	IF IP_C.ERROR > DWORD#0 AND IP_C.C_ENABLE AND NOT IP_C.TIME_RESET THEN  (* IP Control 1 *)
		IF ip_c_red_disable = FALSE OR IP_C.ERROR <> DWORD#16#FD000000 THEN
			ERROR_C := IP_C.ERROR;
			ERROR_T := BYTE#2;
			step := 980;
		END_IF;
	END_IF;

	IF FSD.MODE = BYTE#0 THEN
		IF FSD.ERROR > BYTE#0 THEN
			ERROR_C := BYTE_TO_DWORD(FSD.ERROR);
			ERROR_T := BYTE#4; (* Dateizugriff *)
			step := 980;
		END_IF;
	END_IF;
END_IF;

IF TON_WAIT.Q THEN (* Ablaufstörung - Schrittkette *)
	ERROR_C := SHL(INT_TO_DWORD(step),16) OR INT_TO_DWORD(rcv_state); (* aktuellen Schritt und letzten SMTP Status eintragen *)
	ERROR_T := BYTE#5;
	step := 980;
END_IF;

(* ######################################################## *)

DNS_CLIENT(IP_C:=IP_C, S_BUF:=S_BUF, R_BUF:=R_BUF, DOMAIN:=URL_DATA.DOMAIN, IP4_DNS:= DNS_IP4, ACTIVATE:=step=10); (* DNS-Client *)
IPC(IP:= DWORD#0, PORT:= WORD#0 , TIME_OUT:= TIMEOUT, IP_C:= IP_C, S_BUF:= S_BUF, R_BUF:= R_BUF); (* SMTP Steuerkanal *)
FS(FSD:=FSD,PT:=F_BUF); (* FILE_SERVER *)
BASE64_ENCODE_STR(RUN:= b64_start, STR1:= b64_str1, STR2:= b64_str2, DONE=> b64_done); (* BASE64 kodierung *)

TON_WAIT(IN:=step = last_step AND step > 0,PT:=timeout2);
last_step := step;
activate_last := ACTIVATE;
BUSY := step <> 0;

(* revision history
ks	01. jan. 2011	rev 1.0
	original version
ks	06. apr. 2011	rev 1.1
	list_len und list_get durch element_count und element_get ersetzt
ks	11. may 2011	rev 1.2
	ip_control - remote disconnect error ausblenden, und sonderbehandlung für pcworx
ks	30. may 2011	rev 1.3
	fehler bei receive-timeout
ks	05. may. 2012	rev 1.4
	FileServer AutoClose entfernt und Fehler im Alias Name korrigiert
ks	06. apr. 2013	rev 1.5
	Fehler bei Authorisierungsabfrage bei 1&1 Provider behoben
ks	22. feb. 2016	rev 1.6
	integration SSL/TLS
ks	11. aug. 2016	rev 1.7
	bugfix: Find SSL/TLS String in URL_DATA.PROTOCOL
*)

END_FUNCTION_BLOCK

// POUs/CONVERT/MD5_CRAM_AUTH
FUNCTION_BLOCK MD5_CRAM_AUTH
VAR_IN_OUT
	RUN : BOOL;
	USERNAME : STRING(64);
	PASSWORD : STRING(64);
	B64_TS : STRING(64);  (* Base64 coded ServerTimeStamp *)
	AUTH_KEY : STRING(192);
END_VAR
VAR
	BASE64_DECODE_STR : BASE64_DECODE_STR;
	BASE64_ENCODE_STR : BASE64_ENCODE_STR;
	MD5_STREAM : MD5_STREAM;
	step : INT;
	md5_mode : INT;
	buf : ARRAY [0..63] OF BYTE;
	md5 : ARRAY [0..15] OF BYTE;
	md5_first : ARRAY [0..15] OF BYTE;
	md5_str1 : STRING(64);
	md5_str2 : STRING(64);
	size : UDINT;
	n1 : INT;
	n2 : INT;
	pos : UDINT;
	b64d_run : BOOL;
	b64d_done : BOOL;
	b64e_run : BOOL;
	b64e_done : BOOL;
	str_192 : STRING(192);
	str_144 : STRING(144);
	xpad : BYTE;
	pt : POINTER TO BYTE;
END_VAR

(*
version 1.0		10. may 2010
programmer 	ks
tested by		ks

Der Baustein MD5_CRAM_AUTH (Challenge-Response Authentication Mechanism, Message Digest 5) benutzt
das Authentifizierungsverfahren nach dem Challenge-Response-Prinzip auf der Basis des MD5-HMAC-Algorithmus.
Es wird beispielsweise zur Authentifizierung gegenüber SMTP- oder IMAP-Servern eingesetzt, da es die Übertragung des Passworts im Klartext vermeidet.
Durch dieses Verfahren kann auch über unverschlüsselte Kanäle eine sichere Authentifizierung gegenüber einem Server erfolgen


*)

CASE step OF

0:	IF RUN THEN
		step := 5;
		str_192 := B64_TS;
		b64d_run := TRUE;
	END_IF;

5: IF B64D_DONE THEN (* IPAD Zyklus *)
		b64d_run := FALSE;
		xpad := 16#36;
		md5_str1 := PASSWORD;
		md5_str2 := str_144;
		size := 64 + LEN(md5_str2);
		md5_mode := 1;
		step := 10;
	END_IF;

10: IF md5_mode = 3 THEN (* OPAD Zyklus *)
		md5_first := md5; (* md5 array vom IPAD sichern *)
		xpad := 16#5C;
		size := 64 + 16;
		md5_mode := 1;
		step := 20;
	END_IF;

20: IF md5_mode = 3 THEN
		md5_mode := 0;
		str_144 := CONCAT(USERNAME , ' ');
		str_144 := CONCAT(str_144 , MD5_TO_STRH(md5));
		b64e_run := TRUE;
		step := 30;
	END_IF;

30: IF B64E_DONE THEN
		AUTH_KEY := str_192;
		b64e_run := FALSE;
		RUN := FALSE;
		step := 0; (* alles beendet !! *)
	END_IF;

END_CASE;

(* ----------- md5 -------------- *)
CASE md5_mode OF

1:	n2 := LEN(md5_str1) - 1;
	pt := ADR(md5_str1);
	FOR n1 := 0 TO n2 DO (* string in buf kopieren *)
		buf[n1] := pt^ XOR xpad;
		pt := pt + 1;
	END_FOR;
	FOR n1 := n2 + 1 TO 63 DO (* mit ipad füllen *)
		buf[n1] := xpad;
	END_FOR;

2:	(* Data copy and Calc *)
	IF size > 0 AND pos >= 64 THEN
		IF step = 20 THEN
			FOR n1 := 0 TO 15 DO
				buf[n1] := md5_first[n1];
			END_FOR;
		ELSE
			n2 := LEN(md5_str2) - 1;
			pt := ADR(md5_str2);
			FOR n1 := 0 TO n2 DO (* string in buf kopieren *)
				buf[n1] := pt^;
				pt := pt + 1;
			END_FOR;
		END_IF;
	END_IF;

END_CASE;

IF md5_mode > 0 THEN
	MD5_STREAM(SIZE:=size, MODE:=md5_mode, BUF:=buf, MD5:=md5, POS=>pos);
END_IF;

BASE64_DECODE_STR(RUN:=b64d_run, STR1:=str_192, STR2:=str_144, DONE=>b64d_done);
BASE64_ENCODE_STR(RUN:=b64e_run, STR1:=str_144, STR2:=str_192, DONE=>b64e_done);

(* revision history

hm		10. mai. 2010	rev 1.0
	original version
*)

END_FUNCTION_BLOCK

// POUs/CONVERT/MD5_TO_STRH
FUNCTION MD5_TO_STRH : STRING(32)
VAR_INPUT
	MD5 : ARRAY [0..15] OF BYTE;
END_VAR
VAR
	i : INT;
	tmp : BYTE;
	pt : POINTER TO BYTE;
END_VAR
(*
version 1.0	06. dec. 2009
programmer 	ks
tested BY	ks

MD5_TO_STRH konvertiert das MD5 Hash Array in einen HEX-String
*)

pt := ADR(MD5_TO_STRH); (* read output adress to pointer *)

FOR i := 0 TO 15 DO; (* write the 8 hex characters backwards *)
	tmp := SHR(MD5[i],4);
	PT^ := tmp + SEL(tmp <= 9,87,48);
	pt := pt + 1; (* decrement the pointer *)
	tmp := MD5[i] AND 2#1111;
	PT^ := tmp + SEL(tmp <= 9,87,48);
	pt := pt + 1; (* decrement the pointer *)
END_FOR;
pt^:= 0; (* write the closing byte for the string *)

(* revision history

ks	6. dec. 2009 rev 1.0
	original version

*)

END_FUNCTION

// POUs/CONVERT/MD5_STREAM
FUNCTION_BLOCK MD5_STREAM
VAR_IN_OUT
	MODE : INT;
	BUF : ARRAY [0..63] OF BYTE;
	MD5 : ARRAY [0..15] OF BYTE;
	SIZE : UDINT;
END_VAR

VAR_OUTPUT
	POS : UDINT;
END_VAR

VAR
	hash : ARRAY [0..3] OF DWORD;
	a : DWORD;
	b : DWORD;
	c : DWORD;
	d : DWORD;
	end : UDINT;
	block : UDINT;
	x : ARRAY [0..15] OF DWORD;
	n : INT;
	n1 : INT;
	z : INT;
	pad_1 : BOOL;
END_VAR

(*
version 1.0	06. dec. 2009
programmer 	ks
tested BY	ks

MD5_STREAM berechnet den MD5 Hash eines Datenstromes
*)

CASE MODE OF

1:	(* Initialisierung der Hash-Werte *)
	hash[0] := DWORD#16#67452301;
	hash[1] := DWORD#16#EFCDAB89;
	hash[2] := DWORD#16#98BADCFE;
	hash[3] := DWORD#16#10325476;

	block := SHR(SIZE,6) + BOOL_TO_UDINT((UDINT_TO_BYTE(SIZE) AND 16#3F) > 55);
	pad_1 := FALSE;
	POS := 0;
	End := SIZE;
	SIZE := MIN(64,End);
	MODE := 2;

2:	(* Fuell-Bytes anhängen *)
	FOR n := UDINT_TO_INT(SIZE) TO 63 DO
		BUF[n] := 0;
	END_FOR;

	IF SIZE < 64 AND NOT pad_1 THEN
		BUF[SIZE] := 2#1000_0000;
		pad_1 := TRUE;
	END_IF;

	POS := POS + SIZE;
	SIZE := MIN(64,End - POS);

	n := 0;	(* Byte-Array in DWORD-Array umkopieren *)
	FOR n1 := 0 TO 15 DO
		x[n1] := OSCAT_BASIC.DWORD_OF_BYTE(BUF[n+3],BUF[n+2],BUF[n+1],BUF[n]); (* Little Endian Format *)
		n := n + 4;
	END_FOR;

	IF block = 0 THEN (* am Ende des letzten Blocks die Datenlänge eintragen *)
		x[14] := SHL(UDINT_TO_DWORD(End),3); (* Anzahl Datenbits im Little-Endian Format eintragen *)
		MODE := 3;
	ELSE
		block := block - 1;
	END_IF;

	a := hash[0];
	b := hash[1];
	c := hash[2];
	d := hash[3];

	a := MD5_AUX(1, a, b, c, d, X[00], 07, 16#D76AA478); (* 01 *)
	d := MD5_AUX(1, d, a, b, c, X[01], 12, 16#E8C7B756); (* 02 *)
	c := MD5_AUX(1, c, d, a, b, X[02], 17, 16#242070DB); (* 03 *)
	b := MD5_AUX(1, b, c, d, a, X[03], 22, 16#C1BDCEEE); (* 04 *)
	a := MD5_AUX(1, a, b, c, d, X[04], 07, 16#F57C0FAF); (* 05 *)
	d := MD5_AUX(1, d, a, b, c, X[05], 12, 16#4787C62A); (* 06 *)
	c := MD5_AUX(1, c, d, a, b, X[06], 17, 16#A8304613); (* 07 *)
	b := MD5_AUX(1, b, c, d, a, X[07], 22, 16#FD469501); (* 08 *)
	a := MD5_AUX(1, a, b, c, d, X[08], 07, 16#698098D8); (* 09 *)
	d := MD5_AUX(1, d, a, b, c, X[09], 12, 16#8B44F7AF); (* 10 *)
	c := MD5_AUX(1, c, d, a, b, X[10], 17, 16#FFFF5BB1); (* 11 *)
	b := MD5_AUX(1, b, c, d, a, X[11], 22, 16#895CD7BE); (* 12 *)
	a := MD5_AUX(1, a, b, c, d, X[12], 07, 16#6B901122); (* 13 *)
	d := MD5_AUX(1, d, a, b, c, X[13], 12, 16#FD987193); (* 14 *)
	c := MD5_AUX(1, c, d, a, b, X[14], 17, 16#A679438E); (* 15 *)
	b := MD5_AUX(1, b, c, d, a, X[15], 22, 16#49B40821); (* 16 *)

	a := MD5_AUX(2, a, b, c, d, X[01], 05, 16#F61E2562); (* 17 *)
	d := MD5_AUX(2, d, a, b, c, X[06], 09, 16#C040B340); (* 18 *)
	c := MD5_AUX(2, c, d, a, b, X[11], 14, 16#265E5A51); (* 19 *)
	b := MD5_AUX(2, b, c, d, a, X[00], 20, 16#E9B6C7AA); (* 20 *)
	a := MD5_AUX(2, a, b, c, d, X[05], 05, 16#D62F105D); (* 21 *)
	d := MD5_AUX(2, d, a, b, c, X[10], 09, 16#02441453); (* 22 *)
	c := MD5_AUX(2, c, d, a, b, X[15], 14, 16#D8A1E681); (* 23 *)
	b := MD5_AUX(2, b, c, d, a, X[04], 20, 16#E7D3FBC8); (* 24 *)
	a := MD5_AUX(2, a, b, c, d, X[09], 05, 16#21E1CDE6); (* 25 *)
	d := MD5_AUX(2, d, a, b, c, X[14], 09, 16#C33707D6); (* 26 *)
	c := MD5_AUX(2, c, d, a, b, X[03], 14, 16#F4D50D87); (* 27 *)
	b := MD5_AUX(2, b, c, d, a, X[08], 20, 16#455A14ED); (* 28 *)
	a := MD5_AUX(2, a, b, c, d, X[13], 05, 16#A9E3E905); (* 29 *)
	d := MD5_AUX(2, d, a, b, c, X[02], 09, 16#FCEFA3F8); (* 30 *)
	c := MD5_AUX(2, c, d, a, b, X[07], 14, 16#676F02D9); (* 31 *)
	b := MD5_AUX(2, b, c, d, a, X[12], 20, 16#8D2A4C8A); (* 32 *)

	a := MD5_AUX(3, a, b, c, d, X[05], 04, 16#FFFA3942); (* 33 *)
	d := MD5_AUX(3, d, a, b, c, X[08], 11, 16#8771F681); (* 34 *)
	c := MD5_AUX(3, c, d, a, b, X[11], 16, 16#6D9D6122); (* 35 *)
	b := MD5_AUX(3, b, c, d, a, X[14], 23, 16#FDE5380C); (* 36 *)
	a := MD5_AUX(3, a, b, c, d, X[01], 04, 16#A4BEEA44); (* 37 *)
	d := MD5_AUX(3, d, a, b, c, X[04], 11, 16#4BDECFA9); (* 38 *)
	c := MD5_AUX(3, c, d, a, b, X[07], 16, 16#F6BB4B60); (* 39 *)
	b := MD5_AUX(3, b, c, d, a, X[10], 23, 16#BEBFBC70); (* 40 *)
	a := MD5_AUX(3, a, b, c, d, X[13], 04, 16#289B7EC6); (* 41 *)
	d := MD5_AUX(3, d, a, b, c, X[00], 11, 16#EAA127FA); (* 42 *)
	c := MD5_AUX(3, c, d, a, b, X[03], 16, 16#D4EF3085); (* 43 *)
	b := MD5_AUX(3, b, c, d, a, X[06], 23, 16#04881D05); (* 44 *)
	a := MD5_AUX(3, a, b, c, d, X[09], 04, 16#D9D4D039); (* 45 *)
	d := MD5_AUX(3, d, a, b, c, X[12], 11, 16#E6DB99E5); (* 46 *)
	c := MD5_AUX(3, c, d, a, b, X[15], 16, 16#1FA27CF8); (* 47 *)
	b := MD5_AUX(3, b, c, d, a, X[02], 23, 16#C4AC5665); (* 48 *)

	a := MD5_AUX(4, a, b, c, d, X[00], 06, 16#F4292244); (* 49 *)
	d := MD5_AUX(4, d, a, b, c, X[07], 10, 16#432AFF97); (* 50 *)
	c := MD5_AUX(4, c, d, a, b, X[14], 15, 16#AB9423A7); (* 51 *)
	b := MD5_AUX(4, b, c, d, a, X[05], 21, 16#FC93A039); (* 52 *)
	a := MD5_AUX(4, a, b, c, d, X[12], 06, 16#655B59C3); (* 53 *)
	d := MD5_AUX(4, d, a, b, c, X[03], 10, 16#8F0CCC92); (* 54 *)
	c := MD5_AUX(4, c, d, a, b, X[10], 15, 16#FFEFF47D); (* 55 *)
	b := MD5_AUX(4, b, c, d, a, X[01], 21, 16#85845DD1); (* 56 *)
	a := MD5_AUX(4, a, b, c, d, X[08], 06, 16#6FA87E4F); (* 57 *)
	d := MD5_AUX(4, d, a, b, c, X[15], 10, 16#FE2CE6E0); (* 58 *)
	c := MD5_AUX(4, c, d, a, b, X[06], 15, 16#A3014314); (* 59 *)
	b := MD5_AUX(4, b, c, d, a, X[13], 21, 16#4E0811A1); (* 60 *)
	a := MD5_AUX(4, a, b, c, d, X[04], 06, 16#F7537E82); (* 61 *)
	d := MD5_AUX(4, d, a, b, c, X[11], 10, 16#BD3AF235); (* 62 *)
	c := MD5_AUX(4, c, d, a, b, X[02], 15, 16#2AD7D2BB); (* 63 *)
	b := MD5_AUX(4, b, c, d, a, X[09], 21, 16#EB86D391); (* 64 *)

	hash[0] := hash[0] + a;
	hash[1] := hash[1] + b;
	hash[2] := hash[2] + c;
	hash[3] := hash[3] + d;

END_CASE;

IF MODE = 3 THEN
	z := 0;
	FOR n := 0 TO 3 DO (* von Little-Endian auf Big-Endian format konvertieren und DWORD auf BYTE-Array *)
		FOR n1 := 0 TO 3 DO
			MD5[z] := DWORD_TO_BYTE(hash[n]);
			hash[n] := ROR(hash[n],8);
			z := z + 1;
		END_FOR;
	END_FOR;
END_IF;

(* revision history

ks	6. dec. 2009 rev 1.0
	original version

*)

END_FUNCTION_BLOCK

// POUs/CONVERT/MD5_AUX
FUNCTION MD5_AUX : DWORD
VAR_INPUT
	N : INT;
	A : DWORD;
	B : DWORD;
	C : DWORD;
	D : DWORD;
	X : DWORD;
	U : INT;
	T : DWORD;
END_VAR
VAR
	w : DWORD;
END_VAR

(*
version 1.0	06. dec. 2009
programmer 	ks
tested by	ks

MD5_AUX ist ein Zusatzbaustein füR MD5_STREAM und enthäLT wiederkehrende Berechnungen
*)

CASE N OF
	1: w := (B AND C) OR (NOT(B) AND D);
	2: w := (B AND D) OR (C AND NOT D);
	3: w := (B XOR C XOR D);
	4: w := (C XOR (B OR  NOT(D)));
END_CASE

MD5_AUX := B + ROL(A + w + X + T,U);

(* revision history

ks	6. dec. 2009 rev 1.0
	original version

*)

END_FUNCTION

// POUs/DEMO/DLOG_FILE_HTML_DEMO
PROGRAM DLOG_FILE_HTML_DEMO
VAR
	cur_dt: DT;
	enable: BOOL := TRUE;
	trig_t : TIME := T#5s;
	trig_m : BOOL;
	error_c: DWORD;
	error_t: BYTE;
	auto_close: TIME := T#10s;

	x1: DLOG_DT;
	x2 : DLOG_REAL;
	x3 : DLOG_DINT;
	x4 : DLOG_BOOL;
	x5: DLOG_STRING;
	x : DLOG_DATA;
	RTC_2: oscat_basic.RTC_2;
	DLOG_STORE_FILE_HTML: DLOG_STORE_FILE_HTML;
	GEN_SIN_1: oscat_basic.GEN_SIN;
	COUNT_DR: oscat_basic.COUNT_DR;

	html_caption: STRING := 'Das ist der Titel';
	html_tr_even: STRING := 'BGCOLOR=#B3B7FF';
	html_tr_odd: STRING := 'BGCOLOR=#E0E0E0';
	html_tr_head: STRING := 'BGCOLOR=#FFFF40';
	html_table : STRING := 'BORDER="1"';
END_VAR

VAR RETAIN
	save_data : DLOG_SAVE;
END_VAR
VAR // added by the converter: edge detectors and wires of the graphical bodies
    _w1 : ANY;
END_VAR

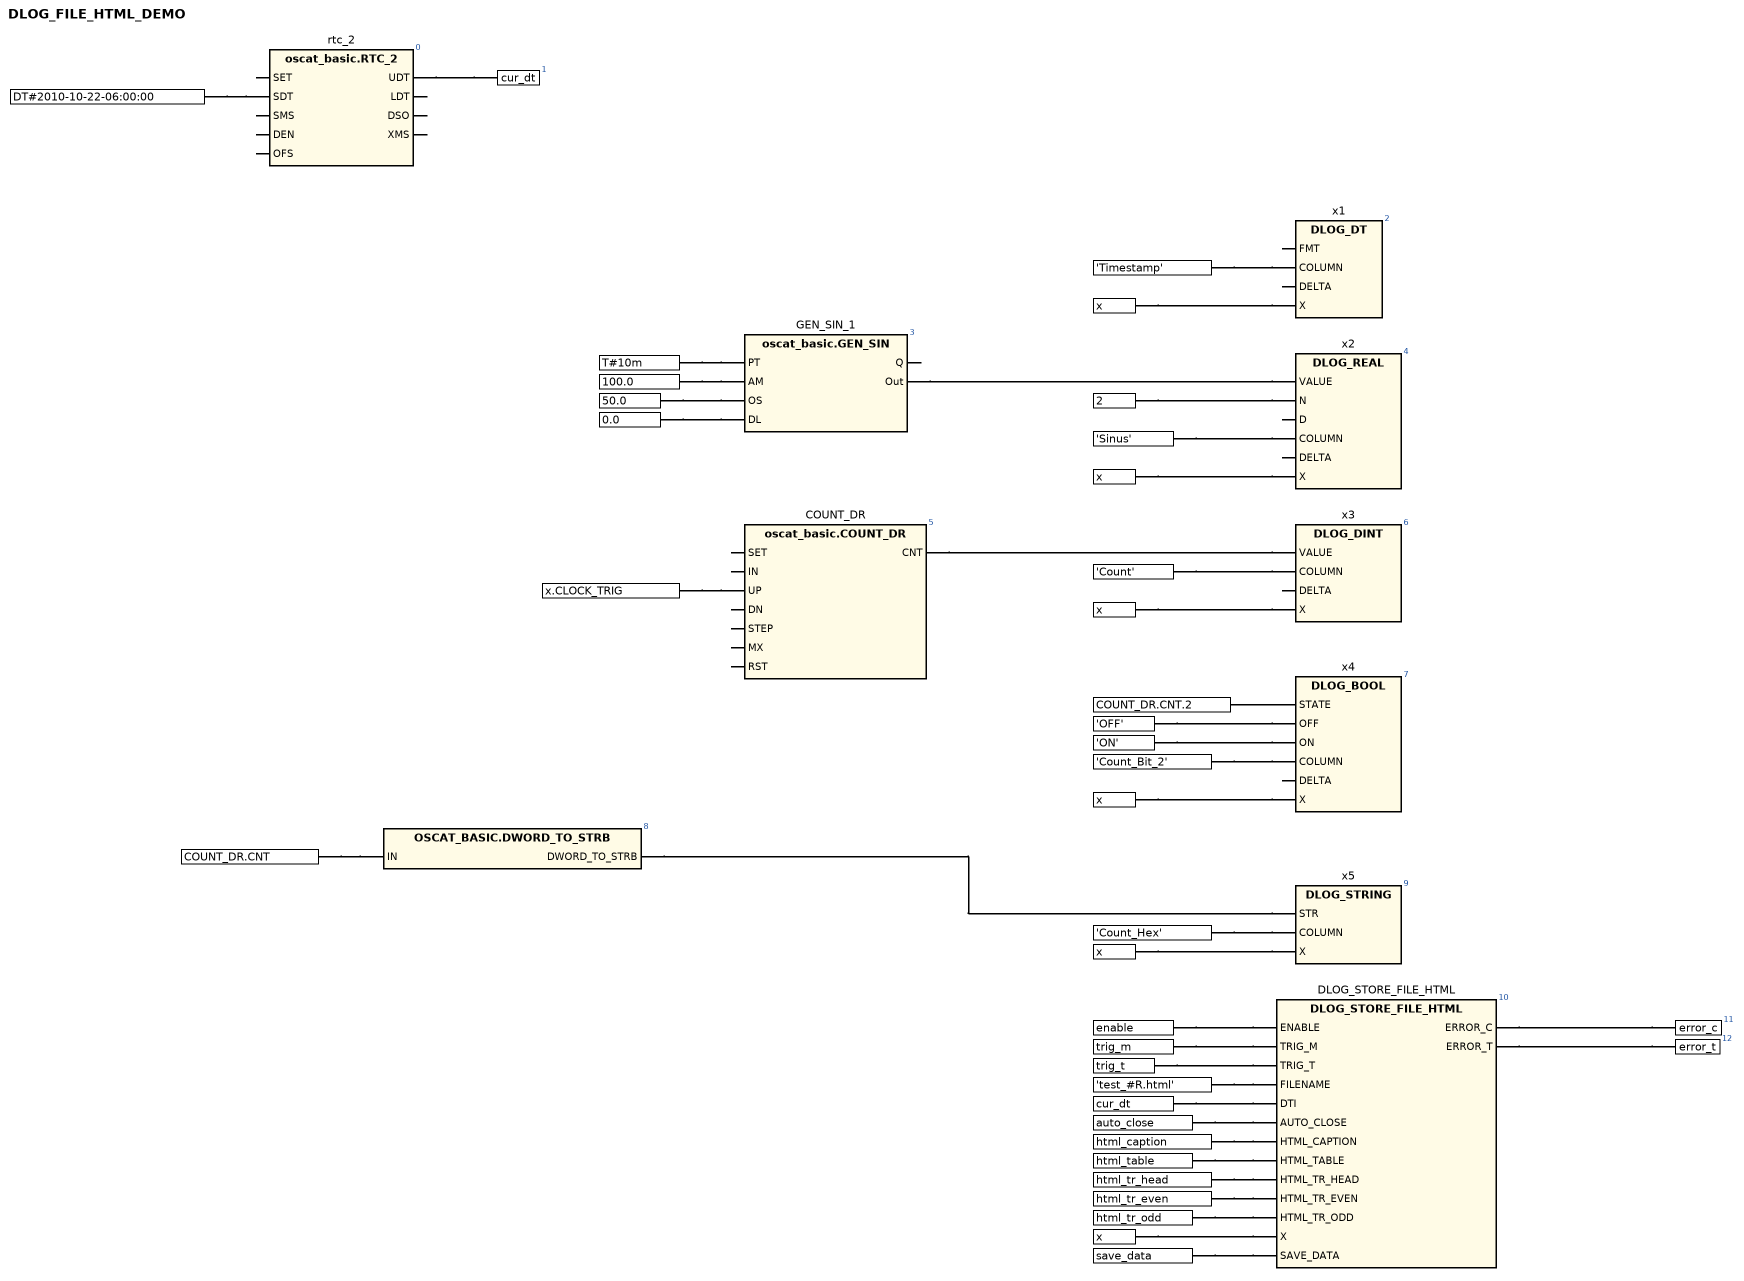
rtc_2(SDT := DT#2010-10-22-06:00:00); // oscat_basic.RTC_2
cur_dt := rtc_2.UDT;
x1(COLUMN := 'Timestamp', X := x); // DLOG_DT
GEN_SIN_1(PT := T#10m, AM := 100.0, OS := 50.0, DL := 0.0); // oscat_basic.GEN_SIN
x2(VALUE := GEN_SIN_1.Out, N := 2, COLUMN := 'Sinus', X := x); // DLOG_REAL
COUNT_DR(UP := x.CLOCK_TRIG); // oscat_basic.COUNT_DR
x3(VALUE := COUNT_DR.CNT, COLUMN := 'Count', X := x); // DLOG_DINT
x4(STATE := COUNT_DR.CNT.2, OFF := 'OFF', ON := 'ON', COLUMN := 'Count_Bit_2', X := x); // DLOG_BOOL
_w1 := OSCAT_BASIC.DWORD_TO_STRB(IN := COUNT_DR.CNT);
x5(STR := _w1, COLUMN := 'Count_Hex', X := x); // DLOG_STRING
DLOG_STORE_FILE_HTML(
    ENABLE := enable,
    TRIG_M := trig_m,
    TRIG_T := trig_t,
    FILENAME := 'test_#R.html',
    DTI := cur_dt,
    AUTO_CLOSE := auto_close,
    HTML_CAPTION := html_caption,
    HTML_TABLE := html_table,
    HTML_TR_HEAD := html_tr_head,
    HTML_TR_EVEN := html_tr_even,
    HTML_TR_ODD := html_tr_odd,
    X := x,
    SAVE_DATA := save_data);
error_c := DLOG_STORE_FILE_HTML.ERROR_C;
error_t := DLOG_STORE_FILE_HTML.ERROR_T;

END_PROGRAM

// POUs/DATA_LOG/DLOG_STORE_FILE_HTML
FUNCTION_BLOCK DLOG_STORE_FILE_HTML
VAR_IN_OUT
	X : DLOG_DATA;
	SAVE_DATA : DLOG_SAVE;
END_VAR
VAR_INPUT
	ENABLE : BOOL;
	TRIG_M : BOOL;
	TRIG_T : TIME;
	FILENAME : STRING;
	DTI : DT;
	AUTO_CLOSE : TIME := T#15s;
	HTML_CAPTION : STRING;
	HTML_TABLE : STRING;
	HTML_TR_HEAD : STRING;
	HTML_TR_EVEN : STRING;
	HTML_TR_ODD : STRING;
END_VAR
VAR_OUTPUT
	ERROR_C : DWORD;
	ERROR_T : BYTE;
END_VAR
VAR
	FS : FILE_SERVER;
	FSD : FILE_SERVER_DATA;
	PT : NETWORK_BUFFER;
	UCB : UNI_CIRCULAR_BUFFER;
	trig_auto : BOOL;
	trig_stored : BOOL;
	trig_tmp : BOOL;
	trig_m_last : BOOL;
	dti_last : DT := DT#2070-02-06-06:28:15;
	fn_last : STRING;
	str : STRING(OSCAT_BASIC.STRING_LENGTH);
	fn : STRING;
	step_1 : INT;
	step_2 : INT;
	idx : INT;
	log_state : USINT;
	log_stop : BOOL;
	n : INT;
	wd_ton : TON;
	wd_time : TIME;
	aw_ton : TON;
	aw_enable : BOOL;
	aw_aktiv : BOOL;
	total_bytes : UDINT;
	cur_ode : BYTE;

	(*
	LOG_MSG : LOG_MSG;
	_debug_enable : BOOL := TRUE;
	*)

END_VAR

(*
version 1.3		21. mar. 2016
programmer		ks
tested by			ks

DLOG_STORE_FILE_HTML schreibt die DLOG Parameter in einen lokale Datei im HMTL-Format 

*)

X.DTI := DTI; (* Datum / Zeit eintragen *)
X.CLOCK_TRIG := DTI <> dti_last;
dti_last := DTI;
trig_auto := FALSE;
IF X.CLOCK_TRIG THEN (* Impuls in jeder Sekunde *)
	fn := OSCAT_BASIC.DT_TO_STRF(DTI, 0, FILENAME, 0); (* automatische Dateinamen generierung *)
	IF TRIG_T >= T#1000ms THEN (* automatischer Trigger *)
		trig_auto := DT_TO_UDINT(DTI) MOD (TIME_TO_UDINT(TRIG_T) / UDINT#1000) = UDINT#0;
	END_IF;
END_IF;

CASE step_1 OF

00:	IF ENABLE THEN
		aw_enable := AUTO_CLOSE >= T#5s;
		wd_time := SEL(X.LOAD_TIME_MAX > T#0s, T#5ms,X.LOAD_TIME_MAX);
		fn_last := fn; (* aktuellen Dateinnamen speichern *)
		IF X.ID_MAX = USINT#0 THEN (* nur einmal nach Satellitenbausteinen scannen *)
			X.ADD_COM := 01; (* ADD INFO *)
			X.STORE_TYPE := BYTE#4; (* HTML-Modus *)
		END_IF;
		step_1 := 10;

		(* ---------------- Debug-Message -----------------------*)
		(*IF _debug_enable THEN
			LOG_CL.NEW_MSG := 'FILE_HTML1 - Start: File [~1], [~2]';
			LOG_CL.PRINTF[1] := fn_last;
			LOG_CL.PRINTF[2] := DT_TO_STRING(DTI);
			LOG_MSG();
		END_IF;*)
		(* -----------------------------------------------------------------*)

	END_IF;

10:	X.UCB.D_STRING := fn_last;
	IF fn_last = SAVE_DATA.FN_REM THEN
		X.UCB.D_HEAD := WORD#16#F201; (* Filemode open + write *)
		X.ADD_COM := 00;
	ELSE
		X.UCB.D_HEAD := WORD#16#F301; (* Filemode create + write *)
		X.ADD_COM := 02; (* ADD HEADER *)
	END_IF;

	X.UCB.D_MODE := 1; (* Dateinamen als String ablegen *)
	UCB(DATA:=X.UCB); (* Daten eintragen *)
	step_1 := 30;

30:	(* LOG-Trigger verarbeiten *)
	trig_tmp := (TRIG_M AND NOT trig_m_last) OR trig_auto OR X.ADD_DATA_REQ;

	IF ENABLE = FALSE OR fn <> fn_last THEN (* ENABLE = 0 oder neuen Dateinamen -> Log Stop *)
		trig_stored := trig_tmp; (* aktuellen Triggerpuls speichern *)
		X.UCB.D_HEAD := WORD#16#EE00;
		X.UCB.D_MODE := 1;
		UCB(DATA:=X.UCB); (* Element schreiben *)
		X.ADD_COM := 00;
		step_1 := 00;

		(* ---------------- Debug-Message -----------------------*)
		(*IF _debug_enable THEN
			LOG_CL.NEW_MSG := 'FILE_HTML1 - Stop: [~2]';
			LOG_CL.PRINTF[2] := DT_TO_STRING(DTI);
			LOG_MSG();
		END_IF;*)
		(* -----------------------------------------------------------------*)

	ELSIF ENABLE THEN
		IF trig_tmp OR trig_stored THEN (* manueller, automatischer oder externer Trigger *)
			trig_stored := FALSE;
			X.ADD_COM := 03; (* ADD DATA *)
			SAVE_DATA.TRIG_CNT := SAVE_DATA.TRIG_CNT + UDINT#1;
			SAVE_DATA.TRIG_CNT_TOTAL  := SAVE_DATA.TRIG_CNT_TOTAL + UDINT#1;
			(* ---------------- Debug-Message -----------------------*)
			(*IF _debug_enable THEN
				LOG_CL.NEW_MSG := 'FILE_HTML1 - Trig: [~2]';
				LOG_CL.PRINTF[2] := DT_TO_STRING(DTI);
				LOG_MSG();
			END_IF;*)
			(* -----------------------------------------------------------------*)
		ELSE
			X.ADD_COM := 04;	(* ADD DATA REQ *)
		END_IF;
	END_IF;

END_CASE;
X.ADD_DATA_REQ := FALSE; (* externe Anforderung rücksetzen *)

(* ##################################### *)

CASE step_2 OF

00:	aw_ton(IN:= idx > 0 AND aw_enable , PT:= AUTO_CLOSE); (* AutoWrite Timer *)
	IF aw_ton.Q THEN (* Zeitgesteuertes Datenschreiben *)
		aw_aktiv := TRUE;
		step_2 := 10; (* Daten schreiben *)
		(* ---------------- Debug-Message -----------------------*)
		(*IF _debug_enable THEN
			LOG_CL.NEW_MSG := 'FILE_HTML2 - AutoWrite: [~2]';
			LOG_CL.PRINTF[2] := DT_TO_STRING(DTI);
			LOG_MSG();
		END_IF;*)
		(* -----------------------------------------------------------------*)

	ELSE
		wd_ton(IN:= FALSE, PT:= wd_time);
		wd_ton(IN:= TRUE);
		WHILE X.UCB.BUF_COUNT > 0 AND step_2 = 0 AND wd_ton.Q = FALSE DO

			X.UCB.D_MODE := 10;
			UCB(DATA:=X.UCB); (* Element lesen , aber noch nicht entfernen *)

			IF X.UCB.D_HEAD > WORD#16#F000 THEN (* F301 oder F201 *)

				str := CONCAT('<html><body><table ',HTML_TABLE);
		        		str := CONCAT(str,'><caption>');
		        		str := CONCAT(str,HTML_CAPTION);
		        		str := CONCAT(str,'</caption>');

				IF idx + LEN(str) < SIZEOF(PT.BUFFER) THEN (* Platz für Element vorhanden ? *)

					FSD.MODE := WORD_TO_BYTE(SHR(SHL(X.UCB.D_HEAD,4),12)); (* 0X00 -> 000X = 3 create + write / 2 open + write *)
					FSD.OFFSET := UDINT#0; (* Start bei Dateianfang *)
					FSD.FILENAME := X.UCB.D_STRING; (* Dateiname *)
					PT.SIZE := UINT#0;
					SAVE_DATA.FN_REM := FSD.FILENAME; (* aktuellen Dateinamen remanent sichern *)

					X.NEW_FILE := FSD.FILENAME;
					X.NEW_FILE_SIZE := UDINT#0;
					X.NEW_FILE_RTRIG := FALSE;
					step_2 := 20;
	
					(* Headerdaten schreiben *)
					IF FSD.MODE = BYTE#3 THEN
						SAVE_DATA.TRIG_CNT := UDINT#0; (* Datei neu anlegen -> dann zähler reset *)
						SAVE_DATA.COLOR := FALSE;
						SAVE_DATA.HEAD := FALSE;

						OSCAT_BASIC._STRING_TO_BUFFER(STR:=str, POS:=idx, PT:=ADR(PT.BUFFER), SIZE:=SIZEOF(PT.BUFFER));
						idx := idx + LEN(str);
						X.NEW_FILE_SIZE := total_bytes + INT_TO_UDINT(idx);
					END_IF;

					X.UCB.D_MODE := 11;
					UCB(DATA:=X.UCB); (* Element entfernen *)

					(* ---------------- Debug-Message -----------------------*)
					(*IF _debug_enable THEN
						LOG_CL.NEW_MSG := 'FILE_HTML2 - Create: Mode [~1] , [~2]';
						LOG_CL.PRINTF[2] := DT_TO_STRING(DTI);
						LOG_CL.PRINTF[1] := BYTE_TO_STRING(FSD.MODE);
						LOG_MSG();
					END_IF;*)
					(* -----------------------------------------------------------------*)
				END_IF;

			ELSIF X.UCB.D_HEAD = WORD#16#EE00 THEN (* LOG_STOP Command *)

				str := '</table></body></html>';

				IF idx + LEN(str) < SIZEOF(PT.BUFFER) THEN (* Platz für Element vorhanden ? *)

					OSCAT_BASIC._STRING_TO_BUFFER(STR:=str, POS:=idx, PT:=ADR(PT.BUFFER), SIZE:=SIZEOF(PT.BUFFER));
					idx := idx + LEN(str);
					log_stop := TRUE;
					step_2 := 10; (* Daten schreiben *)

					X.UCB.D_MODE := 11;
					UCB(DATA:=X.UCB); (* Element entfernen *)
				END_IF;

			ELSIF idx + LEN(X.UCB.D_STRING) + 120 < SIZEOF(PT.BUFFER) THEN (* Platz für Element vorhanden ? *)

				(* ---------------- Debug-Message -----------------------*)
				(*IF _debug_enable THEN
					LOG_CL.NEW_MSG := 'FILE_CSV2 - BUF: TXT [~1],Pos [~2], [~3]';
					LOG_CL.PRINTF[1] := X.UCB.D_STRING;
					LOG_CL.PRINTF[2] := INT_TO_STRING(idx);
					LOG_CL.PRINTF[3] := DT_TO_STRING(DTI);
					LOG_MSG();
				END_IF;*)
				(* -----------------------------------------------------------------*)

				IF log_state = USINT#0 THEN
					str := '<TR ';
					IF NOT SAVE_DATA.HEAD THEN
						str := CONCAT(str,HTML_TR_HEAD);
						SAVE_DATA.HEAD := TRUE;
					ELSIF SAVE_DATA.COLOR THEN
						str := CONCAT(str,HTML_TR_EVEN);
					ELSE
						str := CONCAT(str,HTML_TR_ODD);
					END_IF;
					str := CONCAT(str,'><TD>');
				ELSE
					str := '<TD>';
				END_IF;

				OSCAT_BASIC._STRING_TO_BUFFER(STR:=str, POS:=idx, PT:=ADR(PT.BUFFER), SIZE:=SIZEOF(PT.BUFFER));
				idx := idx + LEN(str);
				log_state := log_state + USINT#1;

				OSCAT_BASIC._STRING_TO_BUFFER(STR:=X.UCB.D_STRING, POS:=idx, PT:=ADR(PT.BUFFER), SIZE:=SIZEOF(PT.BUFFER));
				idx := idx + LEN(X.UCB.D_STRING);
				n := n + USINT#1;
				IF n >= X.ID_MAX THEN
					n := USINT#0;
					str := '</TD></TR>';
					SAVE_DATA.COLOR := NOT SAVE_DATA.COLOR;
					log_state := USINT#0;
				ELSE
					str := '</TD>';
				END_IF;
				OSCAT_BASIC._STRING_TO_BUFFER(STR:=str, POS:=idx, PT:=ADR(PT.BUFFER), SIZE:=SIZEOF(PT.BUFFER));
				idx := idx + LEN(str);
				X.NEW_FILE_SIZE := total_bytes + INT_TO_UDINT(idx);

				X.UCB.D_MODE := 11;
				UCB(DATA:=X.UCB); (* Element entfernen *)

			ELSE (* kein Platz vorhanden *)
				step_2 := 10; (* Daten schreiben *)

			END_IF;
			wd_ton();
		END_WHILE;
	END_IF;

10:	IF idx > 0 THEN (* Daten schreiben *)
		FSD.MODE := BYTE#2; (* File_Open_Exist + File_Write *)
		FSD.OFFSET := UDINT#4294967294; (* 16#FFFF_FFFE ->Spezialcode: Daten automatisch an Dateiende anhängen *)
		PT.SIZE := INT_TO_UINT(idx); (* Datenlänge eintragen *)
		idx := 0;
		(* ---------------- Debug-Message -----------------------*)
		(*IF _debug_enable THEN
			LOG_CL.NEW_MSG := 'FILE_HTML2 - WriteData: Mode [~3] Size [~1] , [~2]';
			LOG_CL.PRINTF[1] := UINT_TO_STRING(PT.SIZE);
			LOG_CL.PRINTF[2] := DT_TO_STRING(DTI);
			LOG_CL.PRINTF[3] := BYTE_TO_STRING(FSD.MODE);
			LOG_MSG();
		END_IF;*)
		(* -----------------------------------------------------------------*)
	END_IF;
	step_2 := 20;

20:	IF FSD.MODE = BYTE#0 THEN
		total_bytes := FSD.FILE_SIZE;
		X.NEW_FILE_SIZE := total_bytes + INT_TO_UDINT(idx);
		IF log_stop OR aw_aktiv THEN
			aw_aktiv := FALSE;
			FSD.MODE := BYTE#5; (* Datei schliessen *)
			(* ---------------- Debug-Message -----------------------*)
			(*IF _debug_enable THEN
				LOG_CL.NEW_MSG := 'FILE_HTML2 - Close: [~2]';
				LOG_CL.PRINTF[2] := DT_TO_STRING(DTI);
				LOG_MSG();
			END_IF;*)
			(* -----------------------------------------------------------------*)
		END_IF;
		step_2 := 30;
	END_IF;

30:	IF FSD.MODE = BYTE#0 THEN (* Datei schliessen beendet *)
		IF log_stop THEN
			X.NEW_FILE_RTRIG := TRUE;
			log_stop := FALSE;
			SAVE_DATA.FN_REM := ''; (* remanenten Dateinamen löschen *)
		END_IF;
		step_2 := 00;
	END_IF;

END_CASE;

FS(FSD:=FSD,PT:=PT); (* FILE_SERVER *)

(* Fehlerauswertung *)
IF FSD.ERROR <> BYTE#0 THEN
	ERROR_C := BYTE_TO_DWORD(FSD.ERROR);
	ERROR_T := BYTE#1;
ELSIF X.UCB.BUF_DATA_LOST > UDINT#0 THEN
	ERROR_C := DWORD#2; (* Fehler: Bufferüberlauf - Datenmenge reduzieren *)
	ERROR_T := BYTE#6; 	(* Type: Buffer *)
ELSIF X.UCB.BUF_USED_MAX > USINT#90 THEN
	ERROR_C := DWORD#1; (* Warnung: Buffer auslastung > 90% *)
	ERROR_T := BYTE#6;	(* Type: Buffer *)
ELSE
	ERROR_C := DWORD#0;
	ERROR_T := BYTE#0;
END_IF;

trig_m_last := TRIG_M;

(* revision history
ks	25. july. 2011	rev 1.0
	original version

ks	16. apr. 2012	rev 1.1
	neuer überarbeiteter Code für automatisches File-open/close

ks	8. mar. 2016	rev 1.2
	nur einmal nach satellitenbausteinen scannen

ks	21. mar. 2016	rev 1.3
	prüfung auf freien bufferplatz hinzugefügt
	fehlermeldungen hinzugefügt

*)

END_FUNCTION_BLOCK

// POUs/DEMO/DLOG_FILE_XML_DEMO
PROGRAM DLOG_FILE_XML_DEMO
VAR
	cur_dt: DT;
	enable: BOOL := TRUE;
	trig_t : TIME := T#5s;
	trig_m : BOOL;
	error_c: DWORD;
	error_t: BYTE;
	auto_close: TIME := T#10s;

	x1: DLOG_DT;
	x2 : DLOG_REAL;
	x3 : DLOG_DINT;
	x4 : DLOG_BOOL;
	x5: DLOG_STRING;
	x : DLOG_DATA;
	RTC_2: oscat_basic.RTC_2;
	DLOG_STORE_FILE_XML: DLOG_STORE_FILE_XML;
	GEN_SIN_1: oscat_basic.GEN_SIN;
	COUNT_DR: oscat_basic.COUNT_DR;
END_VAR

VAR RETAIN
	save_data : DLOG_SAVE;
END_VAR
VAR // added by the converter: edge detectors and wires of the graphical bodies
    _w1 : ANY;
END_VAR

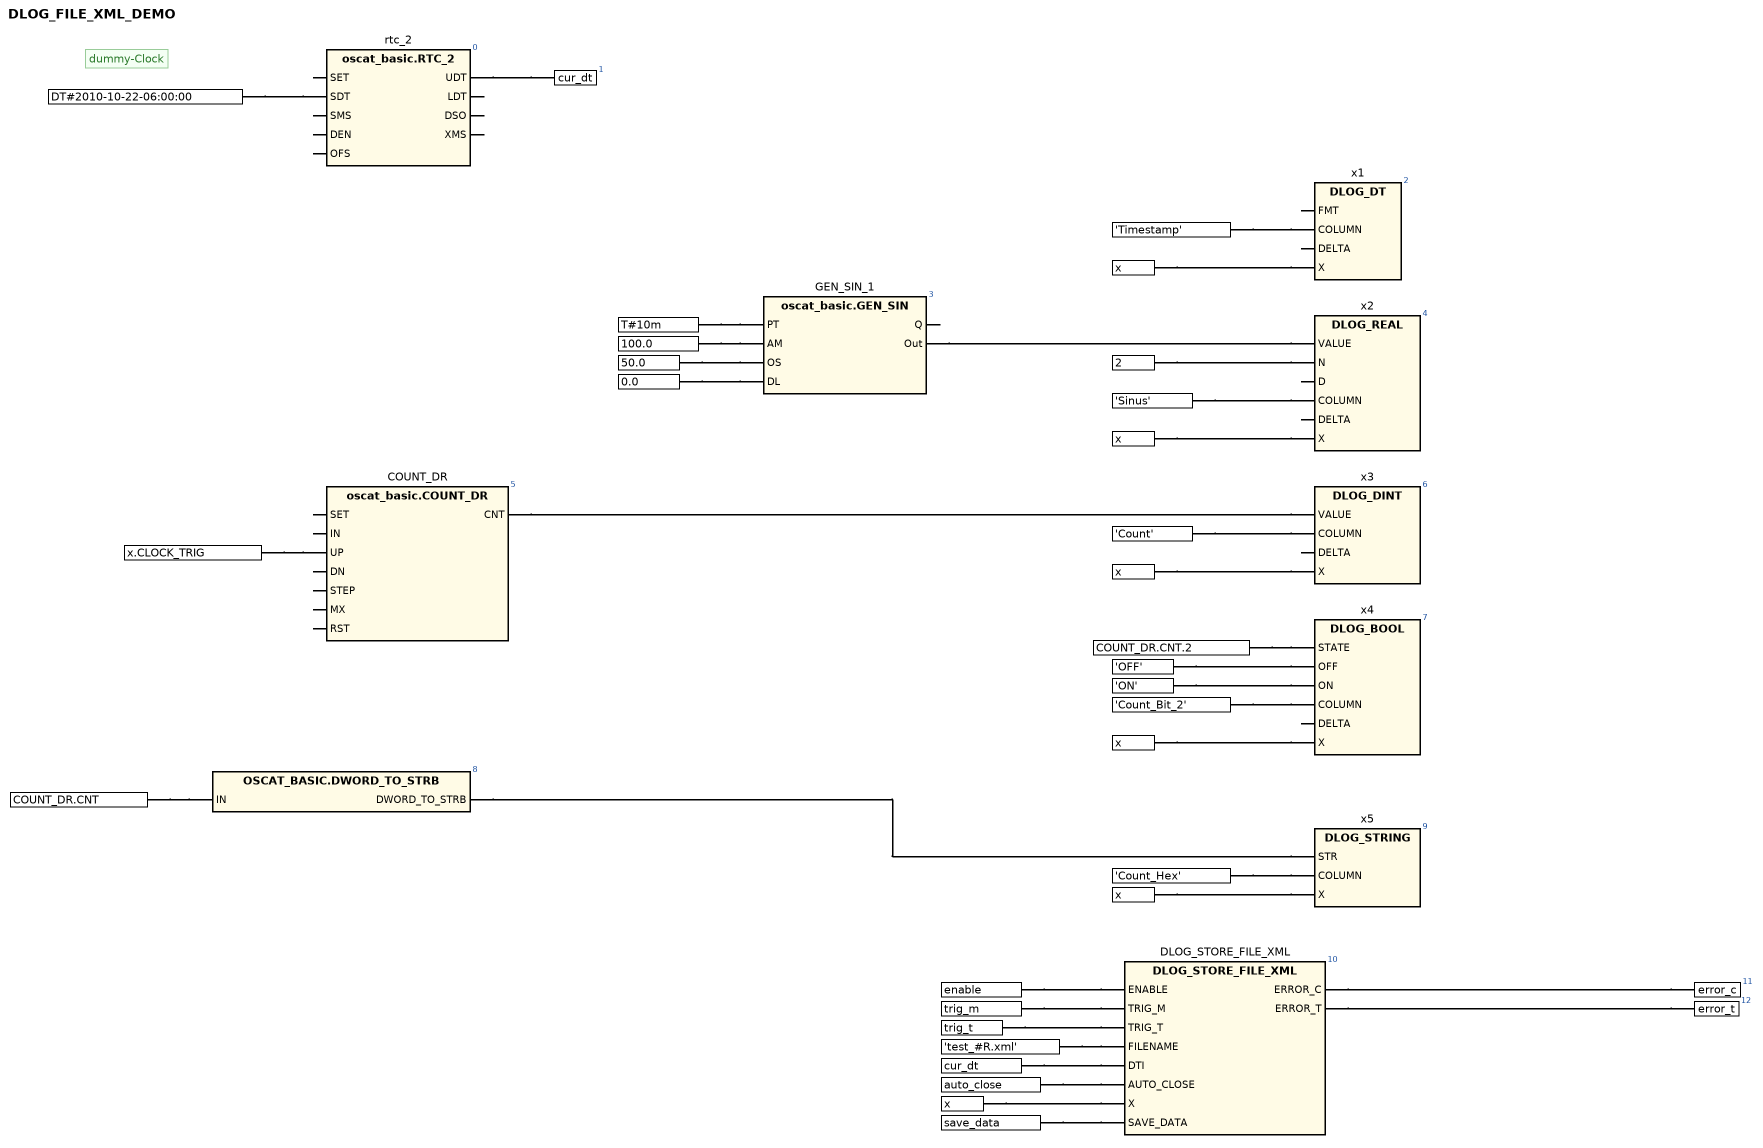
// dummy-Clock
rtc_2(SDT := DT#2010-10-22-06:00:00); // oscat_basic.RTC_2
cur_dt := rtc_2.UDT;
x1(COLUMN := 'Timestamp', X := x); // DLOG_DT
GEN_SIN_1(PT := T#10m, AM := 100.0, OS := 50.0, DL := 0.0); // oscat_basic.GEN_SIN
x2(VALUE := GEN_SIN_1.Out, N := 2, COLUMN := 'Sinus', X := x); // DLOG_REAL
COUNT_DR(UP := x.CLOCK_TRIG); // oscat_basic.COUNT_DR
x3(VALUE := COUNT_DR.CNT, COLUMN := 'Count', X := x); // DLOG_DINT
x4(STATE := COUNT_DR.CNT.2, OFF := 'OFF', ON := 'ON', COLUMN := 'Count_Bit_2', X := x); // DLOG_BOOL
_w1 := OSCAT_BASIC.DWORD_TO_STRB(IN := COUNT_DR.CNT);
x5(STR := _w1, COLUMN := 'Count_Hex', X := x); // DLOG_STRING
DLOG_STORE_FILE_XML(
    ENABLE := enable,
    TRIG_M := trig_m,
    TRIG_T := trig_t,
    FILENAME := 'test_#R.xml',
    DTI := cur_dt,
    AUTO_CLOSE := auto_close,
    X := x,
    SAVE_DATA := save_data);
error_c := DLOG_STORE_FILE_XML.ERROR_C;
error_t := DLOG_STORE_FILE_XML.ERROR_T;

END_PROGRAM

// POUs/DATA_LOG/DLOG_STORE_FILE_XML
FUNCTION_BLOCK DLOG_STORE_FILE_XML
VAR_IN_OUT
	X : DLOG_DATA;
	SAVE_DATA : DLOG_SAVE;
END_VAR
VAR_INPUT
	ENABLE : BOOL;
	TRIG_M : BOOL;
	TRIG_T : TIME;
	FILENAME : STRING;
	DTI : DT;
	AUTO_CLOSE : TIME := T#15s;
END_VAR
VAR_OUTPUT
	ERROR_C : DWORD;
	ERROR_T : BYTE;
END_VAR
VAR
	FS : FILE_SERVER;
	FSD : FILE_SERVER_DATA;
	PT : NETWORK_BUFFER;
	UCB : UNI_CIRCULAR_BUFFER;
	trig_auto : BOOL;
	trig_stored : BOOL;
	trig_tmp : BOOL;
	trig_m_last : BOOL;
	dti_last : DT := DT#2070-02-06-06:28:15;
	fn_last : STRING;
	fn : STRING;
	str : STRING(OSCAT_BASIC.STRING_LENGTH);
	step_1 : INT;
	step_2 : INT;
	idx : INT;
	log_state : USINT;
	log_stop : BOOL;
	n : INT;
	wd_ton : TON;
	wd_time : TIME;
	aw_ton : TON;
	aw_enable : BOOL;
	aw_aktiv : BOOL;
	total_bytes : UDINT;

	(*
	LOG_MSG : LOG_MSG;
	_debug_enable : BOOL := TRUE;
	*)
END_VAR

(*
version 1.3		21.mar. 2016
programmer		ks
tested by			ks

DLOG_STORE_FILE_XML schreibt die DLOG Parameter in einen lokale Datei im XML-Format 

*)

X.DTI := DTI; (* Datum / Zeit eintragen *)
X.CLOCK_TRIG := DTI <> dti_last;
dti_last := DTI;
trig_auto := FALSE;
IF X.CLOCK_TRIG THEN (* Impuls in jeder Sekunde *)
	fn := OSCAT_BASIC.DT_TO_STRF(DTI, 0, FILENAME, 0); (* automatische Dateinamen generierung *)
	IF TRIG_T >= T#1000ms THEN (* automatischer Trigger *)
		trig_auto := DT_TO_UDINT(DTI) MOD (TIME_TO_UDINT(TRIG_T) / UDINT#1000) = UDINT#0;
	END_IF;
END_IF;

CASE step_1 OF

00:	IF ENABLE THEN
		aw_enable := AUTO_CLOSE >= T#5s;
		wd_time := SEL(X.LOAD_TIME_MAX > T#0s, T#5ms,X.LOAD_TIME_MAX);
		fn_last := fn; (* aktuellen Dateinnamen speichern *)
		IF X.ID_MAX = USINT#0 THEN (* nur einmal nach Satellitenbausteinen scannen *)
			X.ADD_COM := 01; (* ADD INFO *)
			X.STORE_TYPE := BYTE#3; (* XML-Modus *)
		END_IF;
		step_1 := 10;

		(* ---------------- Debug-Message -----------------------*)
		(*IF _debug_enable THEN
			LOG_CL.NEW_MSG := 'FILE_XML1 - Start: File [~1], [~2]';
			LOG_CL.PRINTF[1] := fn_last;
			LOG_CL.PRINTF[2] := DT_TO_STRING(DTI);
			LOG_MSG();
		END_IF;*)
		(* -----------------------------------------------------------------*)

	END_IF;

10:	X.UCB.D_STRING := fn_last;
	IF fn_last = SAVE_DATA.FN_REM THEN
		X.UCB.D_HEAD := WORD#16#F201; (* Filemode open + write *)
		X.ADD_COM := 00;
	ELSE
		X.UCB.D_HEAD := WORD#16#F301; (* Filemode create + write *)
		X.ADD_COM := 02; (* ADD HEADER *)
	END_IF;

	X.UCB.D_MODE := 1; (* Dateinamen als String ablegen *)
	UCB(DATA:=X.UCB); (* Daten eintragen *)
	step_1 := 30;

30:	(* LOG-Trigger verarbeiten *)
	trig_tmp := (TRIG_M AND NOT trig_m_last) OR trig_auto OR X.ADD_DATA_REQ;

	IF ENABLE = FALSE OR fn <> fn_last THEN (* ENABLE = 0 oder neuen Dateinamen -> Log Stop *)
		trig_stored := trig_tmp; (* aktuellen Triggerpuls speichern *)
		X.UCB.D_HEAD := WORD#16#EE00;
		X.UCB.D_MODE := 1;
		UCB(DATA:=X.UCB); (* Element schreiben *)
		X.ADD_COM := 00;
		step_1 := 00;

		(* ---------------- Debug-Message -----------------------*)
		(*IF _debug_enable THEN
			LOG_CL.NEW_MSG := 'FILE_XML1 - Stop: [~2]';
			LOG_CL.PRINTF[2] := DT_TO_STRING(DTI);
			LOG_MSG();
		END_IF;*)
		(* -----------------------------------------------------------------*)

	ELSIF ENABLE THEN
		IF trig_tmp OR trig_stored THEN (* manueller, automatischer oder externer Trigger *)
			trig_stored := FALSE;
			X.ADD_COM := 03; (* ADD DATA *)
			SAVE_DATA.TRIG_CNT := SAVE_DATA.TRIG_CNT + UDINT#1;
			SAVE_DATA.TRIG_CNT_TOTAL  := SAVE_DATA.TRIG_CNT_TOTAL + UDINT#1;
			(* ---------------- Debug-Message -----------------------*)
			(*IF _debug_enable THEN
				LOG_CL.NEW_MSG := 'FILE_XML1 - Trig: [~2]';
				LOG_CL.PRINTF[2] := DT_TO_STRING(DTI);
				LOG_MSG();
			END_IF;*)
			(* -----------------------------------------------------------------*)
		ELSE
			X.ADD_COM := 04;	(* ADD DATA REQ *)
		END_IF;
	END_IF;

END_CASE;
X.ADD_DATA_REQ := FALSE; (* externe Anforderung rücksetzen *)

(* ##################################### *)

CASE step_2 OF

00:	aw_ton(IN:= idx > 0 AND aw_enable , PT:= AUTO_CLOSE); (* AutoWrite Timer *)
	IF aw_ton.Q THEN (* Zeitgesteuertes Datenschreiben *)
		aw_aktiv := TRUE;
		step_2 := 10; (* Daten schreiben *)
		(* ---------------- Debug-Message -----------------------*)
		(*IF _debug_enable THEN
			LOG_CL.NEW_MSG := 'FILE_XML2 - AutoWrite: [~2]';
			LOG_CL.PRINTF[2] := DT_TO_STRING(DTI);
			LOG_MSG();
		END_IF;*)
		(* -----------------------------------------------------------------*)

	ELSE
		wd_ton(IN:= FALSE, PT:= wd_time);
		wd_ton(IN:= TRUE);
		WHILE X.UCB.BUF_COUNT > 0 AND step_2 = 0 AND wd_ton.Q = FALSE DO

			X.UCB.D_MODE := 10;
			UCB(DATA:=X.UCB); (* Element lesen , aber noch nicht entfernen *)

			IF X.UCB.D_HEAD > WORD#16#F000 THEN (* F301 oder F201 *)

				str := '<?xml version="1.0" encoding="UTF-8"?><table>';

				IF idx + LEN(str) < SIZEOF(PT.BUFFER) THEN (* Platz für Element vorhanden ? *)

					FSD.MODE := WORD_TO_BYTE(SHR(SHL(X.UCB.D_HEAD,4),12)); (* 0X00 -> 000X = 3 create + write / 2 open + write *)
					FSD.OFFSET := UDINT#0; (* Start bei Dateianfang *)
					FSD.FILENAME := X.UCB.D_STRING; (* Dateiname *)
					PT.SIZE := UINT#0;
					SAVE_DATA.FN_REM := FSD.FILENAME; (* aktuellen Dateinamen remanent sichern *)

					X.NEW_FILE := FSD.FILENAME;
					X.NEW_FILE_SIZE := UDINT#0;
					X.NEW_FILE_RTRIG := FALSE;
					step_2 := 20;
	
					(* Headerdaten schreiben *)
					IF FSD.MODE = BYTE#3 THEN
						SAVE_DATA.TRIG_CNT := UDINT#0; (* Datei neu anlegen -> dann zähler reset *)

						OSCAT_BASIC._STRING_TO_BUFFER(STR:=str, POS:=idx, PT:=ADR(PT.BUFFER), SIZE:=SIZEOF(PT.BUFFER));
						idx := idx + LEN(str);
						X.NEW_FILE_SIZE := total_bytes + INT_TO_UDINT(idx);
					END_IF;

					X.UCB.D_MODE := 11;
					UCB(DATA:=X.UCB); (* Element entfernen *)

					(* ---------------- Debug-Message -----------------------*)
					(*IF _debug_enable THEN
						LOG_CL.NEW_MSG := 'FILE_XML2 - Create: Mode [~1] , [~2]';
						LOG_CL.PRINTF[2] := DT_TO_STRING(DTI);
						LOG_CL.PRINTF[1] := BYTE_TO_STRING(FSD.MODE);
						LOG_MSG();
					END_IF;*)
					(* -----------------------------------------------------------------*)
				END_IF;

			ELSIF X.UCB.D_HEAD = WORD#16#EE00 THEN (* LOG_STOP Command *)

				str := '</table>';

				IF idx + LEN(str) < SIZEOF(PT.BUFFER) THEN (* Platz für Element vorhanden ? *)

					OSCAT_BASIC._STRING_TO_BUFFER(STR:=str, POS:=idx, PT:=ADR(PT.BUFFER), SIZE:=SIZEOF(PT.BUFFER));
					idx := idx + LEN(str);
					log_stop := TRUE;
					step_2 := 10; (* Daten schreiben *)

					X.UCB.D_MODE := 11;
					UCB(DATA:=X.UCB); (* Element entfernen *)

				END_IF;

			ELSIF idx + LEN(X.UCB.D_STRING) + 120 < SIZEOF(PT.BUFFER) THEN (* Platz für Element vorhanden ? *)

				(* ---------------- Debug-Message -----------------------*)
				(*IF _debug_enable THEN
					LOG_CL.NEW_MSG := 'FILE_XML2 - BUF: TXT [~1],Pos [~2], [~3]';
					LOG_CL.PRINTF[1] := X.UCB.D_STRING;
					LOG_CL.PRINTF[2] := INT_TO_STRING(idx);
					LOG_CL.PRINTF[3] := DT_TO_STRING(DTI);
					LOG_MSG();
				END_IF;*)
				(* -----------------------------------------------------------------*)

				IF log_state = USINT#0 THEN
					str := '<row><entry>';
				ELSE
					str := '<entry>';
				END_IF;

				OSCAT_BASIC._STRING_TO_BUFFER(STR:=str, POS:=idx, PT:=ADR(PT.BUFFER), SIZE:=SIZEOF(PT.BUFFER));
				idx := idx + LEN(str);
				log_state := log_state + USINT#1;

				OSCAT_BASIC._STRING_TO_BUFFER(STR:=X.UCB.D_STRING, POS:=idx, PT:=ADR(PT.BUFFER), SIZE:=SIZEOF(PT.BUFFER));
				idx := idx + LEN(X.UCB.D_STRING);

				n := n + USINT#1;
				IF n >= X.ID_MAX THEN
					n := USINT#0;
					str := '</entry></row>';
					log_state := USINT#0;
				ELSE
					str := '</entry>';
				END_IF;
				OSCAT_BASIC._STRING_TO_BUFFER(STR:=str, POS:=idx, PT:=ADR(PT.BUFFER), SIZE:=SIZEOF(PT.BUFFER));
				idx := idx + LEN(str);
				X.NEW_FILE_SIZE := total_bytes + INT_TO_UDINT(idx);

				X.UCB.D_MODE := 11;
				UCB(DATA:=X.UCB); (* Element entfernen *)

			ELSE (* kein Platz vorhanden *)
				step_2 := 10; (* Daten schreiben *)
			END_IF;
			wd_ton();
		END_WHILE;
	END_IF;

10:	IF idx > 0 THEN (* Daten schreiben *)
		FSD.MODE := BYTE#2; (* File_Open_Exist + File_Write *)
		FSD.OFFSET := UDINT#4294967294; (* 16#FFFF_FFFE ->Spezialcode: Daten automatisch an Dateiende anhängen *)
		PT.SIZE := INT_TO_UINT(idx); (* Datenlänge eintragen *)
		idx := 0;
		(* ---------------- Debug-Message -----------------------*)
		(*IF _debug_enable THEN
			LOG_CL.NEW_MSG := 'FILE_XML2 - WriteData: Mode [~3] Size [~1] , [~2]';
			LOG_CL.PRINTF[1] := UINT_TO_STRING(PT.SIZE);
			LOG_CL.PRINTF[2] := DT_TO_STRING(DTI);
			LOG_CL.PRINTF[3] := BYTE_TO_STRING(FSD.MODE);
			LOG_MSG();
		END_IF;*)
		(* -----------------------------------------------------------------*)
	END_IF;
	step_2 := 20;

20:	IF FSD.MODE = BYTE#0 THEN
		total_bytes := FSD.FILE_SIZE;
		X.NEW_FILE_SIZE := total_bytes + INT_TO_UDINT(idx);
		IF log_stop OR aw_aktiv THEN
			aw_aktiv := FALSE;
			FSD.MODE := BYTE#5; (* Datei schliessen *)
			(* ---------------- Debug-Message -----------------------*)
			(*IF _debug_enable THEN
				LOG_CL.NEW_MSG := 'FILE_XML2 - Close: [~2]';
				LOG_CL.PRINTF[2] := DT_TO_STRING(DTI);
				LOG_MSG();
			END_IF;*)
			(* -----------------------------------------------------------------*)
		END_IF;
		step_2 := 30;
	END_IF;

30:	IF FSD.MODE = BYTE#0 THEN (* Datei schliessen beendet *)
		IF log_stop THEN
			X.NEW_FILE_RTRIG := TRUE;
			log_stop := FALSE;
			SAVE_DATA.FN_REM := ''; (* remanenten Dateinamen löschen *)
		END_IF;
		step_2 := 00;
	END_IF;

END_CASE;

FS(FSD:=FSD,PT:=PT); (* FILE_SERVER *)

(* Fehlerauswertung *)
IF FSD.ERROR <> BYTE#0 THEN
	ERROR_C := BYTE_TO_DWORD(FSD.ERROR);
	ERROR_T := BYTE#1;
ELSIF X.UCB.BUF_DATA_LOST > UDINT#0 THEN
	ERROR_C := DWORD#2; (* Fehler: Bufferüberlauf - Datenmenge reduzieren *)
	ERROR_T := BYTE#6; 	(* Type: Buffer *)
ELSIF X.UCB.BUF_USED_MAX > USINT#90 THEN
	ERROR_C := DWORD#1; (* Warnung: Buffer auslastung > 90% *)
	ERROR_T := BYTE#6;	(* Type: Buffer *)
ELSE
	ERROR_C := DWORD#0;
	ERROR_T := BYTE#0;
END_IF;

trig_m_last := TRIG_M;

(* revision history
ks	25. july. 2011	rev 1.0
	original version

ks	16. apr. 2012	rev 1.1
	neuer überarbeiteter Code für automatisches File-open/close

ks	8. mar. 2016	rev 1.2
	nur einmal nach satellitenbausteinen scannen

ks	21. mar. 2016	rev 1.3
	prüfung auf freien bufferplatz hinzugefügt
	fehlermeldungen hinzugefügt

*)

END_FUNCTION_BLOCK

// POUs/DEMO/DLOG_MYSQL_DEMO
PROGRAM DLOG_MYSQL_DEMO
VAR
	cur_dt: DT;
	enable: BOOL := TRUE;
	trig_t : TIME := T#5s;
	trig_m : BOOL;
	error_c: DWORD;
	error_t: BYTE;

	x1 : DLOG_DT;
	x2 : DLOG_REAL;
	x3 : DLOG_DINT;
	x4 : DLOG_BOOL;
	x5 : DLOG_STRING;
	x : DLOG_DATA;
	mysql_info : MYSQL_INFO;

	RTC_2 : oscat_basic.RTC_2;
	GEN_SIN_1: oscat_basic.GEN_SIN;
	COUNT_DR : oscat_basic.COUNT_DR;

	DLOG_STORE_MYSQL : DLOG_STORE_MYSQL;
	(*url : STRING := 'myuser:mypassword@127.0.0.1';*)
	url : STRING(OSCAT_BASIC.STRING_LENGTH) := 'myuser:mypassword@192.168.178.21';
	db_name : STRING(64) := 'oscat_db';
	tb_name : STRING(64) := 'oscat_tb';
	auto_delete : UDINT := 0;
	timeout : TIME := t#10s;

END_VAR
VAR // added by the converter: edge detectors and wires of the graphical bodies
    _w1, _w2 : ANY;
END_VAR

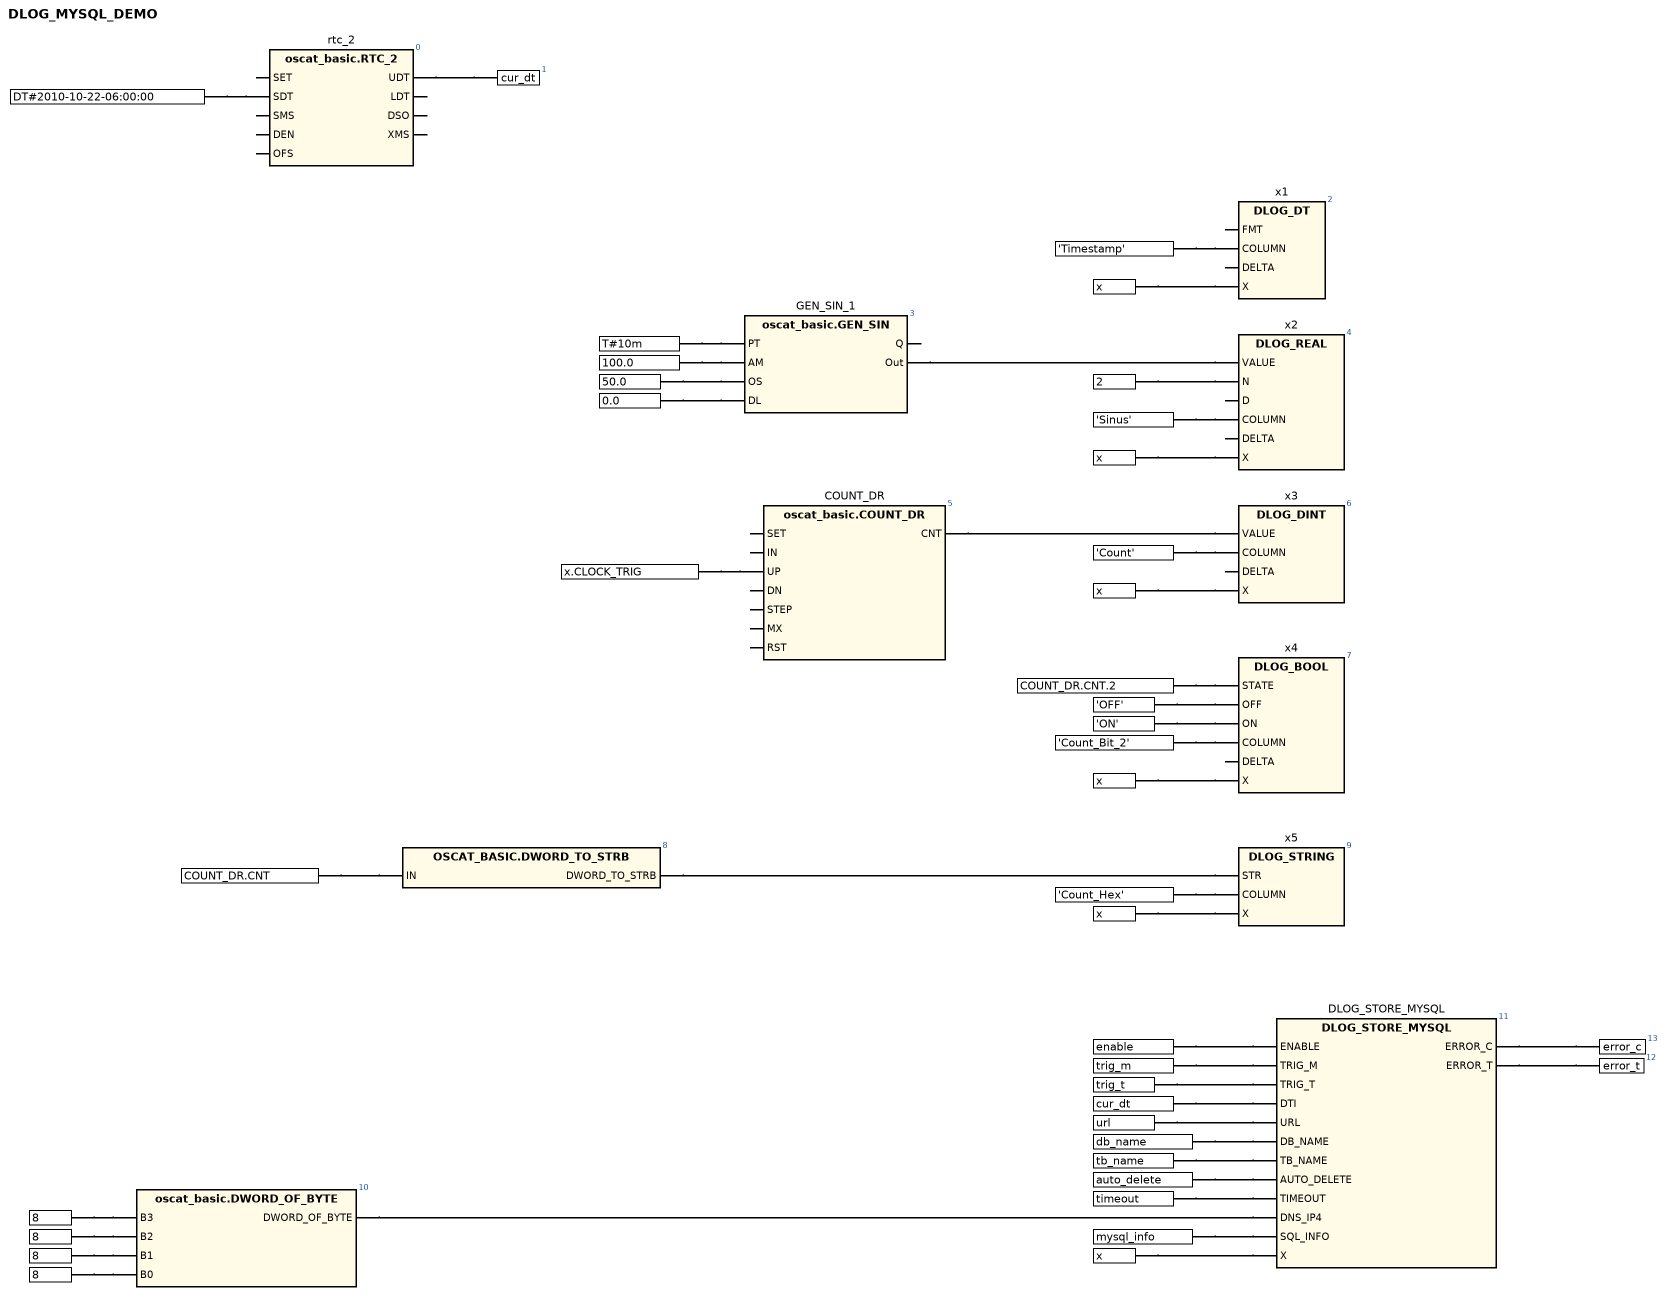
rtc_2(SDT := DT#2010-10-22-06:00:00); // oscat_basic.RTC_2
cur_dt := rtc_2.UDT;
x1(COLUMN := 'Timestamp', X := x); // DLOG_DT
GEN_SIN_1(PT := T#10m, AM := 100.0, OS := 50.0, DL := 0.0); // oscat_basic.GEN_SIN
x2(VALUE := GEN_SIN_1.Out, N := 2, COLUMN := 'Sinus', X := x); // DLOG_REAL
COUNT_DR(UP := x.CLOCK_TRIG); // oscat_basic.COUNT_DR
x3(VALUE := COUNT_DR.CNT, COLUMN := 'Count', X := x); // DLOG_DINT
x4(STATE := COUNT_DR.CNT.2, OFF := 'OFF', ON := 'ON', COLUMN := 'Count_Bit_2', X := x); // DLOG_BOOL
_w1 := OSCAT_BASIC.DWORD_TO_STRB(IN := COUNT_DR.CNT);
x5(STR := _w1, COLUMN := 'Count_Hex', X := x); // DLOG_STRING
_w2 := oscat_basic.DWORD_OF_BYTE(B3 := 8, B2 := 8, B1 := 8, B0 := 8);
DLOG_STORE_MYSQL(
    ENABLE := enable,
    TRIG_M := trig_m,
    TRIG_T := trig_t,
    DTI := cur_dt,
    URL := url,
    DB_NAME := db_name,
    TB_NAME := tb_name,
    AUTO_DELETE := auto_delete,
    TIMEOUT := timeout,
    DNS_IP4 := _w2,
    SQL_INFO := mysql_info,
    X := x);
error_t := DLOG_STORE_MYSQL.ERROR_T;
error_c := DLOG_STORE_MYSQL.ERROR_C;

END_PROGRAM

// POUs/DATA_LOG/DLOG_STORE_MYSQL
FUNCTION_BLOCK DLOG_STORE_MYSQL
VAR_IN_OUT
	SQL_INFO : MYSQL_INFO;
	X : DLOG_DATA;
END_VAR
VAR_INPUT
	ENABLE : BOOL;
	TRIG_M : BOOL;
	TRIG_T : TIME;
	DTI : DT;
	URL : STRING(OSCAT_BASIC.STRING_LENGTH);
	DB_NAME : STRING(64);
	TB_NAME : STRING(64);
	AUTO_DELETE : UDINT;
	TIMEOUT : TIME;
	DNS_IP4 : DWORD;
END_VAR
VAR_OUTPUT
	ERROR_C : DWORD;
	ERROR_T : BYTE;
END_VAR
VAR
	UCB : UNI_CIRCULAR_BUFFER;
	MYSQL_CONTROL: MYSQL_CONTROL;
	trig_auto : BOOL;
	trig_tmp : BOOL;
	trig_m_last : BOOL;
	dti_last : DT := DT#2070-02-06-06:28:15;
	enable_last : BOOL;
	step : INT;
	idx : INT;
	n : USINT;
	snd_text : STRING(OSCAT_BASIC.STRING_LENGTH);
	snd_size : INT;
	sql_command : BYTE;
	next_step : INT;
	i1 : INT;
	i2 : INT;
	y: MYSQL_COM;
	del_dt : UDINT;
	del_start : BOOL;
	run : BOOL;

	(*
	LOG_MSG : LOG_MSG;
	_debug_enable : BOOL := TRUE;
	*)
END_VAR

(*
version 1.3		21. mar. 2016
programmer		ks
tested by			ks

DLOG_STORE_MYSQL der Baustein schreibt die DLOG Parameter in eine MySQL Datenbank
*)

X.DTI := DTI; (* Datum / Zeit eintragen *)
X.CLOCK_TRIG := DTI <> dti_last;
dti_last := DTI;
trig_auto := FALSE;
IF X.CLOCK_TRIG THEN (* Impuls in jeder Sekunde *)
	del_start := DT_TO_UDINT(DTI) - del_dt > AUTO_DELETE AND AUTO_DELETE > UDINT#0;
	IF TRIG_T >= T#1000ms THEN (* automatischer Trigger *)
		trig_auto := DT_TO_UDINT(DTI) MOD (TIME_TO_UDINT(TRIG_T) / UDINT#1000) = UDINT#0;
	END_IF;
END_IF;
X.ADD_COM := 00;

CASE step OF

00:	IF ENABLE AND enable_last = FALSE THEN
		y.SQL_URL := URL;
		y.TIMEOUT := TIMEOUT;
		y.DNS_IP4 := DNS_IP4;
		y.SQL_CON := TRUE;

		X.UCB.D_MODE := 99; (* Buffer reset - Alles löschen *)
		UCB(DATA:=X.UCB);

		IF X.ID_MAX = USINT#0 THEN (* nur einmal nach Satellitenbausteinen scannen *)
			X.ADD_COM := 01; (* ADD INFO *)
			X.STORE_TYPE := BYTE#5; (* MySQL-Modus *)
		END_IF;

		step := 05;
	END_IF;

05:	X.ADD_COM := 02; (* ADD HEADER *)
	step := 10;

10:	IF SQL_INFO.SQL_CONNECTED THEN
		sql_command := BYTE#3; (* CREATE DATABASE IF NOT EXISTS `db_name` *)
		snd_text :=  CONCAT('CREATE DATABASE IF NOT EXISTS `' ,DB_NAME);
		snd_text :=  CONCAT(snd_text, '`');
		next_step := 20;
	END_IF;

20:	sql_command := BYTE#2; (* 0x02 COM_INIT_DB mysql_select_db *)
	snd_text := DB_NAME;
	next_step := 30;

30:	(* CREATE TABLE IF NOT EXISTS tb_name (Timestamp TIMESTAMP NULL DEFAULT CURRENT_TIMESTAMP, n1,n2) *)
	sql_command := BYTE#0;
	idx := 5;
	n := USINT#0;
	WHILE sql_command = BYTE#0 DO
		IF n = USINT#0 THEN
			snd_text := CONCAT('CREATE TABLE IF NOT EXISTS `', TB_NAME);
			snd_text := CONCAT(snd_text,'` (`ID` BIGINT NOT NULL AUTO_INCREMENT PRIMARY KEY ,');
			snd_text := CONCAT(snd_text,' store_timestamp TIMESTAMP NULL DEFAULT CURRENT_TIMESTAMP');
		ELSIF n <= X.ID_MAX THEN
			X.UCB.D_MODE := 12; (* Element lesen und löschen *)
			UCB(DATA:=X.UCB);
			snd_text := CONCAT(', `',X.UCB.D_STRING);
			CASE WORD_TO_INT(SHR(X.UCB.D_HEAD,8)) OF
			02:	snd_text := CONCAT(snd_text, '` FLOAT'); (* REAL *)
			06:	snd_text := CONCAT(snd_text, '` BOOL'); (* BOOL *)
			08:	snd_text := CONCAT(snd_text, '` INT'); (* DINT *)
			13:	snd_text := CONCAT(snd_text, '` DATETIME'); (* DT *)
			ELSE
				snd_text := CONCAT(snd_text, '` VARCHAR(80)'); (* STRING(80) *)
			END_CASE;
		ELSE
			snd_text := ')';
			sql_command := BYTE#3;
			snd_size := idx + LEN(snd_text);
			next_step := 40;
		END_IF;
		OSCAT_BASIC._STRING_TO_BUFFER(str:=snd_text,pos:=idx,pt:=ADR(y.S_BUF.BUFFER),size:=SIZEOF(y.S_BUF.BUFFER)); (* String in puffer kopieren *)
		idx := idx + LEN(snd_text);
		n := n + USINT#1;

		(*####################  DEBUG-MESSAGE  ###################################*)
		(*IF _debug_enable THEN
			LOG_CL.NEW_MSG := 'dlog_mysql: create >~1<';
			LOG_CL.PRINTF[1] := snd_text;
			LOG_MSG();
		END_IF;*)
		(*########################################################################*)
	END_WHILE;

40:	IF del_start THEN
		del_start := FALSE;
		sql_command := BYTE#3; (* DELETE FROM `tb_name` WHERE TIMESTAMPDIFF(SECOND, Timestamp, NOW()) > xxx *)
		snd_text := CONCAT('DELETE FROM `', TB_NAME);
		snd_text := CONCAT(snd_text, '` WHERE TIMESTAMPDIFF(SECOND, store_timestamp, NOW()) > ');
		snd_text := CONCAT(snd_text, UDINT_TO_STRING(AUTO_DELETE));
		next_step := 40;
		del_dt := DT_TO_UDINT(DTI);
		(*####################  DEBUG-MESSAGE  ###################################*)
		(*IF _debug_enable THEN
			LOG_CL.NEW_MSG := 'dlog_mysql: # delete time:~1 >~2<';
			LOG_CL.PRINTF[1] := UDINT_TO_STRING(AUTO_DELETE);
			LOG_CL.PRINTF[2] := snd_text;
			LOG_MSG();
		END_IF;*)
		(*########################################################################*)

         (* INSERT INTO `tb_name` VALUES (CURRENT_TIMESTAMP,  "n1","n2") *)
	ELSIF X.UCB.BUF_COUNT >= USINT_TO_INT(X.ID_MAX) AND step > 0 THEN (* Neue Datenreihe(n) vorhanden *)
		idx := 5;
		n := USINT#0;
		sql_command := BYTE#0;
		WHILE sql_command = BYTE#0 DO
			IF n = USINT#0 THEN
				snd_text := CONCAT('INSERT INTO `', TB_NAME);
				snd_text := CONCAT(snd_text,'` VALUES (NULL, CURRENT_TIMESTAMP');
			ELSIF n <= X.ID_MAX THEN
				X.UCB.D_MODE := 12; (* Element lesen und löschen *)
				UCB(DATA:=X.UCB);
				snd_text := CONCAT(', "',X.UCB.D_STRING);
				snd_text := CONCAT(snd_text, '"');
			ELSE
				snd_text := ')';
				sql_command := BYTE#3;
				snd_size := idx + LEN(snd_text);
				next_step := 40;
			END_IF;
			OSCAT_BASIC._STRING_TO_BUFFER(str:=snd_text,pos:=idx,pt:=ADR(y.S_BUF.BUFFER),size:=SIZEOF(y.S_BUF.BUFFER)); (* String in puffer kopieren *)
			idx := idx + LEN(snd_text);
			n := n + USINT#1;

			(*####################  DEBUG-MESSAGE  ###################################*)
			(*IF _debug_enable THEN
				LOG_CL.NEW_MSG := 'dlog_mysql: insert >~1<';
				LOG_CL.PRINTF[1] := snd_text;
				LOG_MSG();
			END_IF;*)
			(*########################################################################*)
		END_WHILE;
	END_IF;

	IF ENABLE THEN 	(* LOG-Trigger verarbeiten *)
		trig_tmp := (TRIG_M AND NOT trig_m_last) OR trig_auto OR X.ADD_DATA_REQ;

		IF trig_tmp THEN (* manueller, automatischer oder externer Trigger *)
			X.ADD_COM := 03; (* ADD DATA *)
			(* ---------------- Debug-Message -----------------------*)
			(*IF _debug_enable THEN
				LOG_CL.NEW_MSG := 'dlog_mysql: Trigger: DATE [~2]';
				LOG_CL.PRINTF[2] := DT_TO_STRING(DTI);
				LOG_MSG();
			END_IF;*)
			(* -----------------------------------------------------------------*)
		ELSE
			X.ADD_COM := 04;	(* ADD DATA REQ *)
		END_IF;
	ELSE
		y.SQL_CON := FALSE; (* MySQL Verbindung beenden *)
		step := 0;
	END_IF;
	X.ADD_DATA_REQ := FALSE;

(* ~~~~~~~~~~~~~~~~~~~~~~ *)

199:IF y.SQL_RCV_STATE = BYTE#1 THEN (* OK *)
		step := next_step;
	ELSIF y.SQL_RCV_STATE = BYTE#2 THEN  (* FEHLER *)
		step := 0;
	END_IF;

END_CASE;

(* ########################## *)
(* SQL-Kommando ausführen *)
IF sql_command > BYTE#0 THEN

	IF snd_size > 0 THEN
		y.S_BUF.SIZE := INT_TO_UINT(snd_size);
		snd_size := 0;
	ELSE
		OSCAT_BASIC._STRING_TO_BUFFER(str:=snd_text,pos:=5,pt:=ADR(y.S_BUF.BUFFER),size:=SIZEOF(y.S_BUF.BUFFER)); (* String in puffer kopieren *)
		y.S_BUF.SIZE := INT_TO_UINT(5 + LEN(snd_text));
		snd_text := '';
	END_IF;

	IF y.S_BUF.SIZE > SIZEOF(y.S_BUF.BUFFER) THEN (* buffer überlauf erkannt -> Abbruch *)
		y.S_BUF.SIZE := 0;
		sql_command := BYTE#0;
		y.SQL_CON := FALSE; (* MySQL Verbindung beenden *)
		step := 999; (* Dummy-Schritt *)
	ELSE

		i2 := UINT_TO_INT(y.S_BUF.SIZE) - 1; (* alle " zeichen mit ' ersetzen *)
		FOR i1 := 5 TO i2 DO
			IF y.S_BUF.BUFFER[i1] = BYTE#34 THEN
				y.S_BUF.BUFFER[i1] := BYTE#39;
			END_IF;
		END_FOR;
	
		y.S_BUF.BUFFER[4] := sql_command;
		y.SQL_PACKET_NO := BYTE#255;
		sql_command := BYTE#0;
		step := 199;
	END_IF;
END_IF;

(* ########################## *)

MYSQL_CONTROL(COM:= y, INFO:=SQL_INFO);

(* Fehlerauswertung *)
IF step = 999 THEN	(* Buffer überlauf *)
	ERROR_C := DWORD#3; (* Netzwerkbuffer überlauf *)
	ERROR_T := BYTE#6; 	(* Type: Buffer *)
ELSIF y.ERROR_T > BYTE#0 THEN	(* SQL Error *)
	ERROR_C := y.ERROR_C;
	ERROR_T := y.ERROR_T;
	step := 0;
ELSIF X.UCB.BUF_DATA_LOST > UDINT#0 THEN
	ERROR_C := DWORD#2; (* Fehler: Bufferüberlauf - Datenmenge reduzieren *)
	ERROR_T := BYTE#6; 	(* Type: Buffer *)
ELSIF X.UCB.BUF_USED_MAX > USINT#90 THEN
	ERROR_C := DWORD#1; (* Warnung: Buffer auslastung > 90% *)
	ERROR_T := BYTE#6;	(* Type: Buffer *)
ELSE
	ERROR_C := DWORD#0;
	ERROR_T := BYTE#0;
END_IF;



(* ########################## *)

trig_m_last := TRIG_M;
enable_last := ENABLE;
run := step > 0;

(* revision history
ks	20. apr. 2012	rev 1.0
	original version

ks	17. jan. 2014	rev 1.1
	DELTA Error 

ks	8. mar. 2016	rev 1.2
	nur einmal nach satellitenbausteinen scannen

ks	21. mar. 2016	rev 1.3
	prüfung auf bufferüberlauf und fehlermeldungen hinzugefügt

*)

END_FUNCTION_BLOCK

// POUs/DATABASE/MYSQL_CONTROL
FUNCTION_BLOCK MYSQL_CONTROL
VAR_IN_OUT
	COM : MYSQL_COM;
	INFO : MYSQL_INFO;
END_VAR
VAR_OUTPUT
END_VAR
VAR
	IP_C : IP_C;
	URL_DATA : url;
	DNS_CLIENT : DNS_CLIENT;
	IPC : IP_CONTROL;

	step : INT;
	snd_step : INT;
	TON_WAIT : TON;
	last_step : INT;
	idx1 : INT;
	idx2 : INT;
	idx3 : INT;
	dw_tmp : DWORD;
	timeout1 : TIME;
	timeout2 : TIME;
	ip_c_red_disable : BOOL;
	auth_password : STRING(64);
	auth_run : BOOL;
	MYSQL_AUTH : MYSQL_AUTH;
	scramble1_buffer : ARRAY [0..19] OF BYTE;
	scramble2_buffer : ARRAY [0..19] OF BYTE;
	charset_number : BYTE := 16#08;
	max_packet_size : DWORD := 1024;
	client_flags : DWORD := 16#0003_8601;

	(*
	LOG_MSG : LOG_MSG;
	_debug_enable : BOOL := TRUE;
	*)

END_VAR

(*
version 1.1		14. oct. 2013
programmer		ks
tested by		ks

MYSQL_CONTROL führt einen SQL Befehl auf einem MySQL-Server durch 
*)

CASE step OF

00:	IF COM.SQL_CON THEN
		timeout1 := MAX(T#10s,COM.TIMEOUT);
		timeout2 := timeout1 + T#1s;
		INFO.SQL_ERROR := '';
		COM.ERROR_C := DWORD#0;
		COM.ERROR_T := BYTE#0;
		URL_DATA := STRING_TO_URL(STR:=COM.SQL_URL,DEFAULT_PROTOCOL:='',DEFAULT_PATH:='/');
		step := 10;
	END_IF;

10:	IF DNS_CLIENT.DONE THEN
		step := 20;
	ELSIF DNS_CLIENT.ERROR <> DWORD#0 THEN
		COM.ERROR_C := DNS_CLIENT.ERROR;
		COM.ERROR_T := BYTE#1;
		step := 980;
	END_IF;

20:	(* MySQL Steuerkanal einrichten *)
	IF URL_DATA.PORT = WORD#0 THEN
		URL_DATA.PORT := WORD#3306; (* Standard Port *)
	END_IF;
	IP_C.C_PORT := URL_DATA.PORT; (* Portnummer eintragen *)
  	IP_C.C_IP := DNS_CLIENT.IP4; (* IP eintragen *)
  	IP_C.C_MODE := BYTE#0; (* Mode: TCP+ACTIV+PORT *)
  	IP_C.TIME_RESET := TRUE; (* Zeitueberwachung rücksetzen *)
  	IP_C.C_ENABLE := TRUE; (* Verbindungsaufbau freigeben *)
  	IP_C.R_OBSERVE := TRUE; (* Empfangsueberwachung *)
	COM.R_BUF.SIZE := UINT#0;
	COM.SQL_RCV_STATE := BYTE#0;
	step := 30;

30:	IF COM.SQL_RCV_STATE = BYTE#1 THEN
		INFO.SERVER_PROTOCOL_VERSION := COM.R_BUF.BUFFER[4];

		(* ende markierung von string server_version suchen *)
		idx2 := UINT_TO_INT(COM.R_BUF.SIZE) - 1;
		FOR idx1 := 5 TO idx2 DO
			IF COM.R_BUF.BUFFER[idx1] = BYTE#0 THEN EXIT; END_IF;
		END_FOR;
		idx1 := idx1 + 5; (* terminierung und thread-id überspringen *)

		FOR idx2:=0 TO 7 DO	(* Byte 0-7 *)
			scramble1_buffer[idx2] := COM.R_BUF.BUFFER[idx1];
			idx1 := idx1 + 1;
		END_FOR;
		idx1 := idx1 + 1;
		idx2 := idx1 + 1;
		INFO.SERVER_CAPABILITIES := OSCAT_BASIC.WORD_OF_BYTE(COM.R_BUF.BUFFER[idx2], COM.R_BUF.BUFFER[idx1]);
		idx1 := idx1 + 2;
		INFO.SERVER_LANGUAGE := COM.R_BUF.BUFFER[idx1];
		idx1 := idx1 + 1;
		idx2 := idx1 + 1;
		INFO.SERVER_STATUS := OSCAT_BASIC.WORD_OF_BYTE(COM.R_BUF.BUFFER[idx2], COM.R_BUF.BUFFER[idx1]);
		idx1 := idx1 + 15;

		FOR idx2:=8 TO 19 DO	(* Byte 8-19 *)
			scramble1_buffer[idx2] := COM.R_BUF.BUFFER[idx1];
			idx1 := idx1 + 1;
		END_FOR;

		IF INFO.SERVER_PROTOCOL_VERSION < BYTE#10 THEN  (* Error: protocol version zu niedrig *)
			COM.ERROR_T := BYTE#2;
			COM.ERROR_C := DWORD#1;
			step := 980;
		ELSIF URL_DATA.PASSWORD = '' THEN
			step := 50;
		ELSE
			auth_password := URL_DATA.PASSWORD;
			auth_run := TRUE;
			step := 40;
		END_IF;
	END_IF;

40:	MYSQL_AUTH(RUN:= auth_run,PASSWORD:= auth_password ,MESSAGE:= scramble1_buffer,SCRAMBLE:= scramble2_buffer);
	IF NOT auth_run THEN
		step := 50;
	END_IF;

50: (* Client Authentication Packet *)
	(* Byte 0-3 werden später eingetragen *)
	COM.S_BUF.BUFFER[04] := OSCAT_BASIC.BYTE_OF_DWORD(client_flags, BYTE#0); (* client_flags *)
	COM.S_BUF.BUFFER[05] := OSCAT_BASIC.BYTE_OF_DWORD(client_flags, BYTE#1);
	COM.S_BUF.BUFFER[06] := OSCAT_BASIC.BYTE_OF_DWORD(client_flags, BYTE#2);
	COM.S_BUF.BUFFER[07] := OSCAT_BASIC.BYTE_OF_DWORD(client_flags, BYTE#3);
	COM.S_BUF.BUFFER[08] := OSCAT_BASIC.BYTE_OF_DWORD(max_packet_size, BYTE#0); (* max_packet_size *)
	COM.S_BUF.BUFFER[09] := OSCAT_BASIC.BYTE_OF_DWORD(max_packet_size, BYTE#1);
	COM.S_BUF.BUFFER[10] := OSCAT_BASIC.BYTE_OF_DWORD(max_packet_size, BYTE#2);
	COM.S_BUF.BUFFER[11] := OSCAT_BASIC.BYTE_OF_DWORD(max_packet_size, BYTE#3);
	COM.S_BUF.BUFFER[12] := charset_number; (* charset_number *)
	FOR idx1 := 13 TO 35 DO (* 23 bytes filler always 0x00.. *)
		COM.S_BUF.BUFFER[idx1] := BYTE#0;
	END_FOR;
	idx3 := LEN(URL_DATA.USER);
	FOR idx2 :=1 TO idx3 DO
		COM.S_BUF.BUFFER[idx1] := OSCAT_BASIC.CODE(URL_DATA.USER, idx2);
		idx1 := idx1 + 1;
	END_FOR;
	COM.S_BUF.BUFFER[idx1] := BYTE#0; (* String terminierung eintragen *)
	idx1 := idx1 + 1;
	IF LEN(URL_DATA.PASSWORD) = 0 THEN
		COM.S_BUF.BUFFER[idx1] := BYTE#0; (* scramble_buff length *)
	ELSE
		COM.S_BUF.BUFFER[idx1] := BYTE#20; (* scramble_buff length *)
		FOR idx2 :=0 TO 19 DO
			idx1 := idx1 + 1;
			COM.S_BUF.BUFFER[idx1] := scramble2_buffer[idx2];
		END_FOR;
	END_IF;
	COM.S_BUF.SIZE  := INT_TO_UINT(idx1 + 1); (* Sendelänge eintragen *)

	step := 60;

60:	IF COM.SQL_RCV_STATE = BYTE#1 THEN
		INFO.SQL_CONNECTED := TRUE;
		step := 300;
	END_IF;

(* ================================================== *)

300:	step := SEL(COM.SQL_CON,700,310); (* Schritt-Selektion *)

310:	step := 300; (* dummy step *)

(* ================================================== *)

700: (* COM_QUIT *)
	COM.S_BUF.BUFFER[04] := BYTE#1; (* 0x01 COM_QUIT mysql_close *)
	COM.S_BUF.SIZE := UINT#5; (* Sendelänge eintragen *)
	COM.SQL_PACKET_NO := BYTE#255;
	ip_c_red_disable := TRUE;
	step := 710;

710:	IF IP_C.C_STATE = BYTE#0 THEN (* Verbindung durch SQL-Server beendet ? *)
		step := 980;
	END_IF;

(* ================================================== *)

980:IP_C.C_ENABLE := FALSE; (* MYSQL Steuerkanal schliessen *)
	ip_c_red_disable := FALSE;
	INFO.SQL_CONNECTED := FALSE;
	COM.SQL_CON := FALSE;
	COM.S_BUF.SIZE := UINT#0;
	COM.R_BUF.SIZE := UINT#0;
	snd_step := 0;
	step := 990;
	(*####################  DEBUG-MESSAGE  ###################################*)
	(*IF _debug_enable THEN
		LOG_CL.NEW_MSG := 'QUIT: ERROR CODE >~1< TYPE >~2<';
		LOG_CL.PRINTF[1] := DWORD_TO_STRH(COM.ERROR_C);
		LOG_CL.PRINTF[2] := BYTE_TO_STRING(COM.ERROR_T);
		LOG_MSG();
	END_IF;*)
	(*########################################################################*)

990:IF IP_C.C_STATE = BYTE#0 THEN
		step := 0;
	END_IF;

END_CASE;

(* ++++++++++++++++++++++++++++++++++++++++++++++++++++++++++ *)

IF step >= 30 THEN
	IF COM.R_BUF.SIZE >= UINT#3 AND COM.SQL_RCV_STATE = BYTE#0 THEN (* Daten wurden empfangen ? *)
		IF DWORD_TO_UINT(OSCAT_BASIC.DWORD_OF_BYTE(BYTE#0, COM.R_BUF.BUFFER[2], COM.R_BUF.BUFFER[1], COM.R_BUF.BUFFER[0])) + UINT#4 = COM.R_BUF.SIZE THEN
			COM.SQL_PACKET_NO := COM.R_BUF.BUFFER[3];
			IF COM.R_BUF.BUFFER[4] = BYTE#16#FF THEN
				idx2 := 13; (* Error String - Erstes Zeichen *)
				idx3 := UINT_TO_INT(COM.R_BUF.SIZE) - 1; (* Error String - Letztes Zeichen *)
				FOR idx1 := idx2 TO idx3 DO (* alle ' durch ´ ersetzen *)
					IF COM.R_BUF.BUFFER[idx1] = BYTE#39 THEN
						COM.R_BUF.BUFFER[idx1] := BYTE#96;
					END_IF;
				END_FOR;
				INFO.SQL_ERROR := OSCAT_BASIC.BUFFER_TO_STRING(PT:=ADR(COM.R_BUF.BUFFER),SIZE:=COM.R_BUF.SIZE,START:=INT_TO_UINT(idx2),STOP:=INT_TO_UINT(idx3));
				COM.ERROR_T := BYTE#3;
				COM.ERROR_C := OSCAT_BASIC.DWORD_OF_BYTE(BYTE#0,BYTE#0,COM.R_BUF.BUFFER[6], COM.R_BUF.BUFFER[5]);
				COM.SQL_RCV_STATE := BYTE#2;
				COM.R_BUF.SIZE := UINT#0; (* Empfangsbuffer nach Fehler rücksetzen *)
				step := 980;
			ELSE
				COM.SQL_RCV_STATE := BYTE#1;
				IP_C.R_OBSERVE := FALSE;

				(*####################  DEBUG-MESSAGE  ###################################*)
				(*IF _debug_enable THEN
					LOG_CL.NEW_MSG := 'RCV: size >~1<';
					LOG_CL.PRINTF[1] := UINT_TO_STRING(COM.R_BUF.SIZE);
					LOG_MSG();
				END_IF;*)
				(*########################################################################*)
			END_IF;
		END_IF;
	END_IF;
END_IF;

(* automatisches Datensenden *)

CASE snd_step OF

00:	IF step >= 20 AND COM.S_BUF.SIZE > UINT#0 THEN
		dw_tmp := UINT_TO_DWORD(COM.S_BUF.SIZE - UINT#4); (* packet_length *)
		COM.S_BUF.BUFFER[0] := OSCAT_BASIC.BYTE_OF_DWORD(dw_tmp, BYTE#0);
		COM.S_BUF.BUFFER[1] := OSCAT_BASIC.BYTE_OF_DWORD(dw_tmp, BYTE#1);
		COM.S_BUF.BUFFER[2] := 0;
		COM.SQL_PACKET_NO := COM.SQL_PACKET_NO + 1;
		COM.S_BUF.BUFFER[3] := COM.SQL_PACKET_NO;

		IP_C.R_OBSERVE := TRUE;
		COM.R_BUF.SIZE := UINT#0; (* Empfangsbuffer rücksetzen *)
		COM.SQL_RCV_STATE := BYTE#0;

	        (*####################  DEBUG-MESSAGE  ###################################*)
	        (*IF _debug_enable THEN
	          LOG_CL.NEW_MSG := 'SND: size >~1<';
	          LOG_CL.PRINTF[1] := UINT_TO_STRING(COM.S_BUF.SIZE);
	          LOG_MSG();
	        END_IF;*)
	        (*########################################################################*)

		snd_step := 10;
	END_IF;

10:	IF COM.S_BUF.SIZE = UINT#0 THEN (* warten bis alle daten gesendet sind *)
		snd_step := 0;
	END_IF;

END_CASE;

(* Globale Fehlerbehandlung für Haupt-Routine *)
IF COM.ERROR_T = BYTE#0 AND step > 20 THEN (* noch kein Fehler gespeichert und Hauptroutine aktiv *)
	IF IP_C.ERROR > DWORD#0 AND IP_C.C_ENABLE AND NOT IP_C.TIME_RESET THEN  (* IP Control *)
		IF ip_c_red_disable = FALSE OR IP_C.ERROR <> DWORD#16#FD000000 THEN
			COM.ERROR_C := IP_C.ERROR;
			COM.ERROR_T := BYTE#2;
			step := 980;
		END_IF;
	END_IF;
END_IF;

IF TON_WAIT.Q THEN (* Ablaufstörung - Schrittkette *)
	COM.ERROR_C := INT_TO_DWORD(step); (* aktuellen Schritt eintragen *)
	COM.ERROR_T := BYTE#5;
	step := 980;
END_IF;

(* ######################################################## *)

DNS_CLIENT(IP_C:=IP_C, S_BUF:=COM.S_BUF, R_BUF:=COM.R_BUF, DOMAIN:=URL_DATA.DOMAIN, IP4_DNS:= COM.DNS_IP4, ACTIVATE:=step=10); (* DNS-Client *)
IPC(IP:= DWORD#0, PORT:= WORD#0 , TIME_OUT:= timeout1, IP_C:= IP_C, S_BUF:= COM.S_BUF, R_BUF:= COM.R_BUF); (* MYSQL Steuerkanal *)

TON_WAIT(IN:=step = last_step AND step > 0,PT:=timeout2);
last_step := step;

(* revision history
ks	20. apr. 2012	rev 1.0
	original version
ks	14. oct. 2013	rev 1.1
	DNS_CLIENT Fehler durch zugriffskonflikt zwischen dns_client und mySQL auf S_BUF

*)

END_FUNCTION_BLOCK

// POUs/DATABASE/MYSQL_AUTH
FUNCTION_BLOCK MYSQL_AUTH
VAR_IN_OUT
	RUN : BOOL;
	PASSWORD : STRING(64);
	MESSAGE : ARRAY [0..19] OF BYTE;
	SCRAMBLE : ARRAY [0..19] OF BYTE;
END_VAR
VAR
	SHA1_STREAM : SHA1_STREAM;
	buf : ARRAY [0..63] OF BYTE;
	sha_mode : INT;
	step : INT;
	size : UDINT;
	pos : UDINT;
	i : INT;
	i2: INT;
	scramble1 : ARRAY [0..19] OF BYTE;
	scramble2 : ARRAY [0..19] OF BYTE;
END_VAR

(*
version 1.0		16. apr. 2012
programmer		ks
tested by		ks

MYSQL_AUTH führt das Passwort-Hashing fuer die Anmeldung bei einem MySQL 4.1 Server durch 
*)

IF NOT RUN THEN RETURN; END_IF;
CASE step OF

0:	CASE sha_mode OF
	0:	sha_mode := 1; (* Initialisierung *)
		size := INT_TO_UDINT(LEN(PASSWORD));
		i2 := UDINT_TO_INT(size) - 1;
		FOR i := 0 TO 63 DO
			IF i <= i2 THEN
				buf[i] := OSCAT_BASIC.CODE(STR:=PASSWORD,POS:=i+1);
			ELSE
				buf[i] := BYTE#0;
			END_IF;
		END_FOR;

	3:	scramble1 := SCRAMBLE;
		sha_mode := 1; (* Initialisierung *)
		size := UDINT#20;
		FOR i := 0 TO 19 DO
			buf[i] := scramble1[i];
		END_FOR;
		step := 10;
	END_CASE;

10:	IF sha_mode = 3 THEN
		sha_mode := 1; (* Initialisierung *)
		scramble2 := SCRAMBLE;
		size := UDINT#40;
		FOR i := 0 TO 19 DO
			buf[i] := message[i];
			buf[i+20] := scramble2[i];
		END_FOR;
		step :=20;
	END_IF;

20:	IF sha_mode = 3 THEN
		sha_mode := 0; (* Stop *)
		FOR i:= 0 TO 19 DO
			SCRAMBLE[i] := SCRAMBLE[i] XOR scramble1[i];
		END_FOR;
		step :=0;
		RUN := FALSE;
	END_IF;
END_CASE;

SHA1_STREAM(SIZE:=size, MODE:=sha_mode, BUF:=buf, SHA1:=SCRAMBLE, POS=>pos);

(* revision history
ks	20. apr. 2012	rev 1.0
	original version

*)

END_FUNCTION_BLOCK

// POUs/CONVERT/SHA1_STREAM
FUNCTION_BLOCK SHA1_STREAM
VAR_IN_OUT
	MODE : INT;
	BUF : ARRAY [0..63] OF BYTE;
	SHA1 : ARRAY [0..19] OF BYTE;
	SIZE : UDINT;
END_VAR

VAR_OUTPUT
	POS : UDINT;
END_VAR

VAR
	hash : ARRAY [0..4] OF DWORD;
	end : UDINT;
	block : UDINT;
	pad_1 : BOOL;
	w : ARRAY [0..79] OF DWORD;
	n : INT;
	n1 : INT;
	a : DWORD;
	b : DWORD;
	c : DWORD;
	d : DWORD;
	e : DWORD;
	f : DWORD;
	k : DWORD;
	x : DWORD;
	z : INT;
END_VAR

(*
version 1.0	06. dec. 2009
programmer 	ks
tested BY	ks

SHA1_STREAM berechnet den SHA1 Hash eines Datenstromes
*)

CASE MODE OF

1:	(* Initialisierung der Hash-Werte *)
	hash[0] := DWORD#16#67452301;
	hash[1] := DWORD#16#EFCDAB89;
	hash[2] := DWORD#16#98BADCFE;
	hash[3] := DWORD#16#10325476;
	hash[4] := DWORD#16#C3D2E1F0;

	(* Buffer initialisieren *)
	FOR n := 16 TO 79 DO
   		w[n] := DWORD#0;
	END_FOR;

	block := SHR(SIZE,6) + BOOL_TO_UDINT((UDINT_TO_BYTE(SIZE) AND 16#3F) > 55);	(* benötigte Blocks errechnen *)

	pad_1 := FALSE;
	POS := 0;
	End := SIZE;
	SIZE := MIN(64,End);
	MODE := 2;

2:	FOR n := UDINT_TO_INT(SIZE) TO 63 DO (* Fuell-Bytes anhängen *)
		BUF[n] := 0;
	END_FOR;

	IF SIZE < 64 AND NOT pad_1 THEN
		BUF[SIZE] := 2#1000_0000;
		pad_1 := TRUE;
	END_IF;

	POS := POS + SIZE;
	SIZE := MIN(64,End - POS);

	n := 0;	(* Byte-Array in DWORD-Array umkopieren *)
	FOR n1 := 0 TO 15 DO
		w[n1] := OSCAT_BASIC.DWORD_OF_BYTE(BUF[n],BUF[n+1],BUF[n+2],BUF[n+3]);
		n := n + 4;
	END_FOR;

	IF block = 0 THEN (* am Ende des letzten Blocks die Datenlänge eintragen *)
		w[15] := SHL(UDINT_TO_DWORD(End),3); (* Anzahl Datenbits eintragen *)
		MODE := 3;
	ELSE
		block := block - 1;
	END_IF;

	FOR n := 16 TO 79 DO (* erweitern der 16 32-bit-Worte auf 80 32-bit-Worte *)
		w[n] := ROL(w[n-3] XOR w[n-8] XOR w[n-14] XOR w[n-16],1);
	END_FOR;

	a := hash[0];
	b := hash[1];
	c := hash[2];
	d := hash[3];
	e := hash[4];

	FOR n := 0 TO 79 DO
		IF n <= 19 THEN
			f := (b AND c) OR (NOT(b) AND d);
			k := DWORD#16#5A827999;
		ELSIF n <= 39 THEN
			f := b XOR c XOR d;
			k := DWORD#16#6ED9EBA1;
		ELSIF n <= 59 THEN
			f := (b AND c) OR (b AND d) OR (c AND d);
			k := DWORD#16#8F1BBCDC;
		ELSE
			f := b XOR c XOR d;
			k := DWORD#16#CA62C1D6;
		END_IF;

		x := ROL(a,5) + f + e + k + w[n];
		e := d;
		d := c;
		c := ROL(b,30);
		b := a;
		a := x;
	END_FOR;

	(* aktuelle Hash-Werte zum letzten Wert addieren *)
	hash[0] := hash[0] + a;
	hash[1] := hash[1] + b;
	hash[2] := hash[2] + c;
	hash[3] := hash[3] + d;
	hash[4] := hash[4] + e;

END_CASE;

IF MODE = 3 THEN
	z := 0;
	FOR n := 0 TO 4 DO (* konvertiere DWORD auf BYTE-Array *)
		FOR n1 := 0 TO 3 DO
			hash[n] := ROL(hash[n],8);
			SHA1[z] := DWORD_TO_BYTE(hash[n]);
			z := z + 1;
		END_FOR;
	END_FOR;
END_IF;

(* revision history

ks	6. dec. 2009 rev 1.0
	original version

*)

END_FUNCTION_BLOCK

// POUs/DATA_LOG/DLOG_REAL_ARRAY
FUNCTION_BLOCK DLOG_REAL_ARRAY
VAR_IN_OUT
	R_ARRAY : DLOG_REAL_ARRAY_DATA;
	X : DLOG_DATA;
END_VAR
VAR_INPUT
	N : INT;
	D : STRING(1);
	R_COUNT : INT;
END_VAR
VAR
	UCB : UNI_CIRCULAR_BUFFER;
	id : WORD;
	idx : INT;
END_VAR

(*
version 1.0		18. mar. 2016
programmer		ks
tested by		ks

DLOG_REAL_ARRAY legt alle REAL-Werte aus einem Array als STRING im FIFO-RING-Buffer ab um diesen mit den Baustein DLOG_STORE_*  aufzuzeichnen

*)

FOR idx := 1 TO R_COUNT DO

	CASE x.ADD_COM OF

	01:	(* ADD INFO *)
		X.ID_MAX := X.ID_MAX + USINT#1;
		id := WORD#16#0201; (* Quelltype REAL , Zieltype STRING *)
		(* automatisch Namen vergeben *)
		IF LEN(R_ARRAY[idx].COLUMN) = 0 THEN
			R_ARRAY[idx].COLUMN := CONCAT('Spalte_',USINT_TO_STRING(X.ID_MAX));
		END_IF;
	02:	(* ADD HEADER *)
		X.UCB.D_STRING := R_ARRAY[idx].COLUMN;
		X.UCB.D_HEAD := id;
		X.UCB.D_MODE := 1;
		UCB(DATA:=X.UCB); (* Daten eintragen *)
	03:	(* ADD DATA *)
		X.UCB.D_STRING := OSCAT_BASIC.REAL_TO_STRF(IN:=R_ARRAY[idx]._value_last,N:=N,D:=D);
		X.UCB.D_HEAD := id;
		X.UCB.D_MODE := 1;
		UCB(DATA:=X.UCB); (* Daten eintragen *)
		R_ARRAY[idx]._delta_last := R_ARRAY[idx]._value_last;
	04:	(* ADD DATA REQ *)
		IF R_ARRAY[idx].DELTA <> 0.0 THEN
			IF R_ARRAY[idx].VALUE <= (R_ARRAY[idx]._delta_last - R_ARRAY[idx].DELTA) OR R_ARRAY[idx].VALUE >= (R_ARRAY[idx]._delta_last + R_ARRAY[idx].DELTA) THEN
				X.ADD_DATA_REQ := TRUE;
				R_ARRAY[idx]._delta_last := R_ARRAY[idx].VALUE;
			END_IF;
		END_IF;
	END_CASE;
	R_ARRAY[idx]._value_last := R_ARRAY[idx].VALUE;

END_FOR;

(* revision history
ks	03. mar. 2016	rev 1.0
	original version

*)

END_FUNCTION_BLOCK

// POUs/DEMO/DLOG_RRD_DEMO
PROGRAM DLOG_RRD_DEMO
VAR
	cur_dt: DT;
	trig_t : TIME := T#50s;
	trig_m : BOOL;

	rrd_error_c : DWORD;
	rrd_error_t : BYTE;
	rrd_enable : BOOL := TRUE;
	(*rrd_url : STRING(OSCAT_BASIC.STRING_LENGTH) := 'http://xxx.com/myhouse/rrd/test_rrd.php?rrd_db=test.rrd&value=';*)
	rrd_url : STRING(OSCAT_BASIC.STRING_LENGTH) := '192.168.178.21/rrd/test_rrd2.php?rrd_db=test.rrd&value=';
	rrd_timeout: TIME := t#5s;

	RTC_2 : oscat_basic.RTC_2;
	DLOG_STORE_RRD : DLOG_STORE_RRD;

	x : DLOG_DATA;
	x1 : DLOG_DINT;
	x2 : DLOG_DINT;
	x3 : DLOG_REAL;
	x4 : DLOG_REAL;
	x5 : DLOG_REAL;
	x6 : DLOG_REAL;
	x7 : DLOG_REAL;

	GEN_SIN_1 : oscat_basic.GEN_SIN;
	GEN_SIN_2 : oscat_basic.GEN_SIN;
	GEN_SIN_3 : oscat_basic.GEN_SIN;
	GEN_RMP_1: oscat_basic.GEN_RMP;
	GEN_RMP_2: oscat_basic.GEN_RMP;
END_VAR
VAR // added by the converter: edge detectors and wires of the graphical bodies
    _w1, _w2, _w3 : ANY;
END_VAR

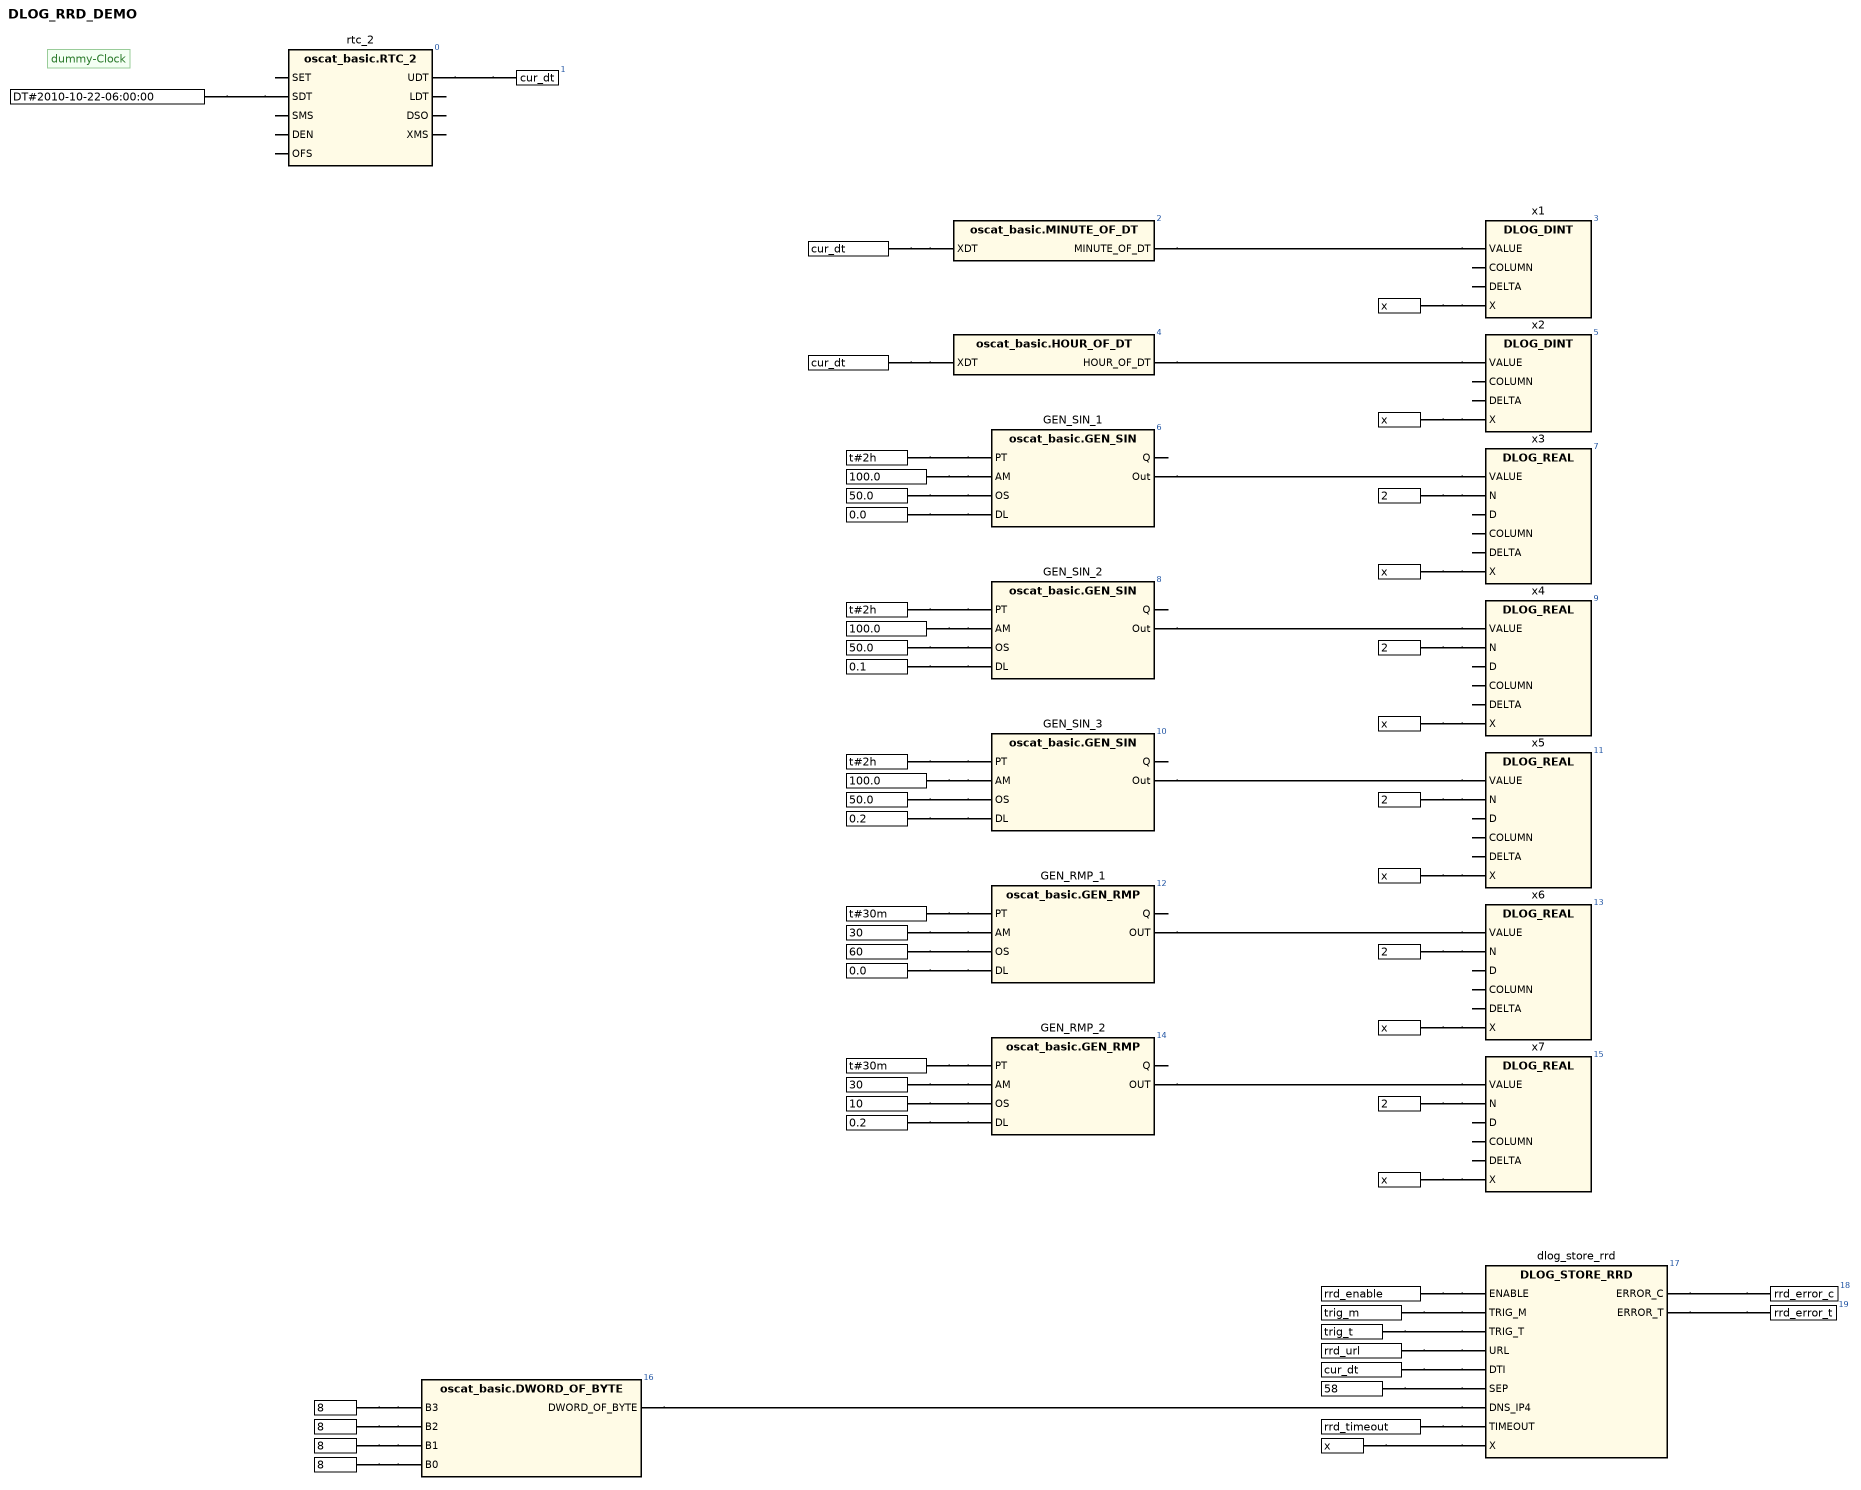
// dummy-Clock
rtc_2(SDT := DT#2010-10-22-06:00:00); // oscat_basic.RTC_2
cur_dt := rtc_2.UDT;
_w1 := oscat_basic.MINUTE_OF_DT(XDT := cur_dt);
x1(VALUE := _w1, X := x); // DLOG_DINT
_w2 := oscat_basic.HOUR_OF_DT(XDT := cur_dt);
x2(VALUE := _w2, X := x); // DLOG_DINT
GEN_SIN_1(PT := t#2h, AM := 100.0, OS := 50.0, DL := 0.0); // oscat_basic.GEN_SIN
x3(VALUE := GEN_SIN_1.Out, N := 2, X := x); // DLOG_REAL
GEN_SIN_2(PT := t#2h, AM := 100.0, OS := 50.0, DL := 0.1); // oscat_basic.GEN_SIN
x4(VALUE := GEN_SIN_2.Out, N := 2, X := x); // DLOG_REAL
GEN_SIN_3(PT := t#2h, AM := 100.0, OS := 50.0, DL := 0.2); // oscat_basic.GEN_SIN
x5(VALUE := GEN_SIN_3.Out, N := 2, X := x); // DLOG_REAL
GEN_RMP_1(PT := t#30m, AM := 30, OS := 60, DL := 0.0); // oscat_basic.GEN_RMP
x6(VALUE := GEN_RMP_1.OUT, N := 2, X := x); // DLOG_REAL
GEN_RMP_2(PT := t#30m, AM := 30, OS := 10, DL := 0.2); // oscat_basic.GEN_RMP
x7(VALUE := GEN_RMP_2.OUT, N := 2, X := x); // DLOG_REAL
_w3 := oscat_basic.DWORD_OF_BYTE(B3 := 8, B2 := 8, B1 := 8, B0 := 8);
dlog_store_rrd(
    ENABLE := rrd_enable,
    TRIG_M := trig_m,
    TRIG_T := trig_t,
    URL := rrd_url,
    DTI := cur_dt,
    SEP := 58,
    DNS_IP4 := _w3,
    TIMEOUT := rrd_timeout,
    X := x);
rrd_error_c := dlog_store_rrd.ERROR_C;
rrd_error_t := dlog_store_rrd.ERROR_T;

END_PROGRAM

// POUs/DATA_LOG/DLOG_STORE_RRD
FUNCTION_BLOCK DLOG_STORE_RRD
VAR_IN_OUT
	X : DLOG_DATA;
END_VAR
VAR_INPUT
	ENABLE : BOOL;
	TRIG_M : BOOL;
	TRIG_T : TIME;
	URL : STRING(OSCAT_BASIC.STRING_LENGTH);
	DTI : DT;
	SEP : BYTE;
	DNS_IP4 : DWORD;
	TIMEOUT : TIME;
END_VAR
VAR_OUTPUT
	ERROR_C : DWORD;
	ERROR_T : BYTE;
END_VAR
VAR
	UCB : UNI_CIRCULAR_BUFFER;
	IP_C : IP_C; (* IP_Control Verwaltungsstruktur *)
	S_BUF : NETWORK_BUFFER;
	R_BUF : NETWORK_BUFFER;
	URL_DATA : url;
	DNS_CLIENT : DNS_CLIENT;
	HTTP_GET : HTTP_GET;
	IPC : IP_CONTROL;

	trig_auto : BOOL;
	trig_stored : BOOL;
	trig_tmp : BOOL;
	trig_m_last : BOOL;
	dti_last : DT := DT#2070-02-06-06:28:15;
	step_1 : INT;
	step_2 : INT;
	sep_char : STRING(1);
	url_query : STRING(OSCAT_BASIC.STRING_LENGTH);
	n : INT;

	(*
	LOG_MSG : LOG_MSG;
	_debug_enable : BOOL := TRUE;
	*)
END_VAR

(*
version 1.4		21. mar. 2016
programmer		ks
tested by			ks

DLOG_STORE_RRD der Baustein übergibt die DLOG Parameter an einen RoundRobinDatabase-Server
*)

X.DTI := DTI; (* Datum / Zeit eintragen *)
X.CLOCK_TRIG := DTI <> dti_last;
dti_last := DTI;
trig_auto := FALSE;
IF X.CLOCK_TRIG THEN (* Impuls in jeder Sekunde *)
	IF TRIG_T >= T#1000ms THEN (* automatischer Trigger *)
		trig_auto := DT_TO_UDINT(DTI) MOD (TIME_TO_UDINT(TRIG_T) / UDINT#1000) = UDINT#0;
	END_IF;
END_IF;

CASE step_1 OF

00:	IF ENABLE THEN
		IF X.ID_MAX = USINT#0 THEN (* nur einmal nach Satellitenbausteinen scannen *)
			X.ADD_COM := 01; (* ADD INFO *)
			X.STORE_TYPE := BYTE#1; (* RRD-Modus *)
		END_IF;

		ERROR_T := BYTE#0;
		ERROR_C := DWORD#0;

		X.UCB.D_MODE := 99;
		UCB(DATA:=X.UCB); (* Buffer löschen *)

		URL_DATA:=STRING_TO_URL(STR:=URL,DEFAULT_PROTOCOL:='',DEFAULT_PATH:=''); (* URL zerlegen *)
		sep_char := OSCAT_BASIC.CHR_TO_STRING(SEP);
		url_query := URL_DATA.QUERY;
		step_1 := 30;

		(* ---------------- Debug-Message -----------------------*)
		(*IF _debug_enable THEN
			LOG_CL.NEW_MSG := 'FILE_RRD1 - Start: DATE [~2]';
			LOG_CL.PRINTF[2] := DT_TO_STRING(DTI);
			LOG_MSG();
		END_IF;*)
		(* -----------------------------------------------------------------*)

	END_IF;

30:	(* LOG-Trigger verarbeiten *)
	trig_tmp := (TRIG_M AND NOT trig_m_last) OR trig_auto OR X.ADD_DATA_REQ;

	IF ENABLE = FALSE THEN (* ENABLE = 0 -> Log Stop *)
		X.ADD_COM := 00;
		step_1 := 00;

		(* ---------------- Debug-Message -----------------------*)
		(*IF _debug_enable THEN
			LOG_CL.NEW_MSG := 'FILE_RRD1 - Stop: DATE [~2]';
			LOG_CL.PRINTF[2] := DT_TO_STRING(DTI);
			LOG_MSG();
		END_IF;*)
		(* -----------------------------------------------------------------*)

	ELSIF ENABLE THEN
		IF trig_tmp OR trig_stored THEN (* manueller, automatischer oder externer Trigger *)
			trig_stored := FALSE;
			X.ADD_COM := 03; (* ADD DATA *)
			(* ---------------- Debug-Message -----------------------*)
			(*IF _debug_enable THEN
				LOG_CL.NEW_MSG := 'FILE_RRD1 - Trig: DATE [~2]';
				LOG_CL.PRINTF[2] := DT_TO_STRING(DTI);
				LOG_MSG();
			END_IF;*)
			(* -----------------------------------------------------------------*)
		ELSE
			X.ADD_COM := 04;	(* ADD DATA REQ *)
		END_IF;
	END_IF;

END_CASE;
X.ADD_DATA_REQ := FALSE; (* externe Anforderung rücksetzen *)

(* ##################################### *)

CASE step_2 OF

00:	IF X.UCB.BUF_DATA_LOST > UDINT#0 THEN
		ERROR_C := DWORD#2; (* Fehler: Bufferüberlauf - Datenmenge reduzieren *)
		ERROR_T := BYTE#6; 	(* Type: Buffer *)
		step_2 := 100;
	ELSIF X.UCB.BUF_USED_MAX > USINT#90 THEN
		ERROR_C := DWORD#1; (* Warnung: Buffer auslastung > 90% *)
		ERROR_T := BYTE#6;	(* Type: Buffer *)
	END_IF;

	IF X.UCB.BUF_COUNT >= USINT_TO_INT(X.ID_MAX) THEN (* genug Einträge vorhanden *)
		URL_DATA.QUERY := url_query; (* original Query wiederherstellen *)
		n := 1;
		WHILE n <= USINT_TO_INT(X.ID_MAX) DO
			X.UCB.D_MODE := 12; (* Element lesen und löschen *)
			UCB(DATA:=X.UCB);
			IF n < USINT_TO_INT(X.ID_MAX) THEN (* Trennzeichen hinzufügen *)
				X.UCB.D_STRING := CONCAT(X.UCB.D_STRING,sep_char);
			END_IF;
			IF LEN(X.UCB.D_STRING) + LEN(URL_DATA.QUERY) <= OSCAT_BASIC.STRING_LENGTH THEN
				URL_DATA.QUERY := CONCAT(URL_DATA.QUERY,X.UCB.D_STRING); (* Query mit LOG-Daten ergänzen *)
				step_2 := 40;
			ELSE
				ERROR_T := BYTE#4; (* LOG-Daten können nicht in URL gepackt werden *)
				ERROR_C := DWORD#1;
				step_2 := 100;
			END_IF;
			n := n + 1;
		END_WHILE;;
	END_IF;

40:	IF DNS_CLIENT.DONE THEN
		step_2 := 60;
	ELSIF (DNS_CLIENT.ERROR > DWORD#0) THEN
		ERROR_C := DNS_CLIENT.ERROR; (* Fehlerbehandlung *)
		ERROR_T := BYTE#1;
		step_2 := 100;
	END_IF;

60:	IF HTTP_GET.DONE THEN
		n := UINT_TO_INT(HTTP_GET.BODY_START);
		IF R_BUF.BUFFER[n] <> BYTE#48 THEN (* ASCII '0' *)
			ERROR_C := DWORD#1;
			ERROR_T := BYTE#3;
		END_IF;
		step_2 := 100;

	ELSIF HTTP_GET.ERROR > DWORD#0 THEN (* Fehlerbehandlung *)
		ERROR_C := HTTP_GET.ERROR;
		ERROR_T := BYTE#2;
		step_2 := 100;
	END_IF;

100:	IF (NOT HTTP_GET.DONE) THEN (* UNLOCK HTTP DATA *)
		step_2 := SEL(ERROR_T = BYTE#0, 120,0);
	END_IF;

120:	IF NOT ENABLE THEN
		step_2 := 0;
	END_IF;

END_CASE;

HTTP_GET(IP_C:=IP_C,S_BUF:=S_BUF,R_BUF:=R_BUF,IP4:=DNS_CLIENT.IP4,GET:=step_2=60,MODE:=2,UNLOCK_BUF:=step_2=100,URL_DATA:=URL_DATA); (* HTTP_GET *)
DNS_CLIENT(IP_C:=IP_C, S_BUF:=S_BUF, R_BUF:=R_BUF, DOMAIN:=URL_DATA.DOMAIN, IP4_DNS:= DNS_IP4, ACTIVATE:=step_2=40); (* DNS-Client *)
IPC(IP:= 0, PORT:= 0 , TIME_OUT:= TIMEOUT, IP_C:= IP_C, S_BUF:= S_BUF, R_BUF:= R_BUF); (* IP_CONTROL *)

trig_m_last := TRIG_M;

(* revision history
ks	01. jan. 2011	rev 1.0
	original version

ks	13. may. 2011	rev 1.1
	ADD_DATA_REQ hinzugefügt

ks	26. july. 2011	rev 1.2
	code optimierung D_MODE 12 und bessere fehlerauswertung

ks	16. apr. 2012	rev 1.3
	neuer überarbeiteter Code

ks	21. mar. 2016	rev 1.4
	nur einmal nach satellitenbausteinen scannen und fehlermeldungen hinzugefügt

*)

END_FUNCTION_BLOCK

// POUs/NETWORK/HTTP_GET
FUNCTION_BLOCK HTTP_GET
VAR_IN_OUT
	URL_DATA : url;
	IP_C : IP_C; (* IP_Control Verwaltungsstruktur *)
	S_BUF : NETWORK_BUFFER;
	R_BUF : NETWORK_BUFFER;
END_VAR
VAR_INPUT
	IP4 : DWORD;
	GET : BOOL;
	MODE : BYTE := BYTE#2;
	UNLOCK_BUF : BOOL;
END_VAR
VAR_OUTPUT
	HTTP_STATUS : STRING;
	HEADER_START : UINT; (* HTTP Header (Message Header) *)
	HEADER_STOP : UINT; (* HTTP Header (Message Header) *)
	BODY_START : UINT; (* Message Body *)
	BODY_STOP : UINT; (* Message Body *)
	DONE : BOOL;
	ERROR : DWORD;
END_VAR
VAR
	READ_HTTP :	READ_HTTP;
	BASE64_ENCODE_STR :	BASE64_ENCODE_STR;
	b64_str1 :	STRING(144);
	b64_str2 :	STRING(192);
	b64_done :	BOOL;
	b64_start :	BOOL;
	authentication :	BOOL;
	IP_FIFO : IP_FIFO;
	ip_state : BYTE;
	ip_id : BYTE;
	get_last : BOOL;
	ip4_stored : DWORD;
	state : INT;
	i : INT;
	http_1_1_host : BOOL;
	total_size : INT;
	text : STRING(OSCAT_BASIC.STRING_LENGTH);
	delimiter2b : STRING(2);
	delimiter4b : STRING(4);
	del_end : STRING(4);
	del_pos : INT;
	idx : INT;
	rcv_timeout : BOOL;
	con_rdce : BOOL;

	(*LOG_MSG : LOG_MSG;
	_debug_enable : BOOL := TRUE;
	_debug_state_last : INT := -1;*)

END_VAR

(*

version 1.4	31. mar. 2016
programmer 	ks
tested by		ks

HTTP_GET führt eine HTTP Abfrage einer Web-Seite bei einem WEB_Server durch, und stellt die Daten ausbereitet zu verfügung




----------------------------------------
Zusatzinfos

D_MODE:

01 Element in Buffer schreiben
10 Element von Buffer lesen, aber nicht entfernen
11 Das zuvor mit Kommando 10 gelesen Element wird entfernt.
12 Element von Buffer lesen, und entfernen
99 Buffer wird rückgesetzt. Alle Daten werden gelöscht

-------------------------------------------------------------

D_HEAD = LEFT-BYTE (ADD-Ino) , RIGHT-BYTE (Type-Kennung)

Type-Kennungen:
1 = STRING (Bei DATA.D_STRING muss der STRING übergeben werden)
2 = REAL (Bei DATA.D_REAL muss der REAL-Wert übergeben werden)
3 = DWORD (Bei DATA.D_DWORD muss das DWORD übergeben werden)

--> alle anderen typekennungen werden als ohne Daten (länge 0) nur als HEAD info abgelegt
X = Header-Information ohne Daten

-------------------------------------------------------------

STORE_CSV

MODE 1 / HEAD F201; schreiben: Filename ablegen + Filemode open + write
MODE 1 / HEAD F301; schreiben: Filemode ablegen + Filemode create + write
MODE 1 / HEAD EE00; schreiben: Log Stop

-------------------------------------------------------------

HEAD
0x0101; Quelltype STRING , Zieltype STRING
0x0201; Quelltype REAL   , Zieltype STRING
0x0601; Quelltype BOOL   , Zieltype STRING
0x0801; Quelltype DINT   , Zieltype STRING
0x0D01; Quelltype DT     , Zieltype STRING

-------------------------------------------------------------

X.STORE_TYPE := BYTE#1; RRD-Modus
X.STORE_TYPE := BYTE#2; CSV-Modus
X.STORE_TYPE := BYTE#3; XML-Modus
X.STORE_TYPE := BYTE#4; HTML-Modus
X.STORE_TYPE := BYTE#5; MySQL-Modus

----------------------------------------------


*)

CASE state OF
00:	DONE := FALSE;
	IF GET AND NOT GET_LAST THEN (* auf positive Flanke SET warten *)
		state := 10;
		ip4_stored := IP4; (* aktuelle IP4 speichern *)
		total_size := 0;
		HEADER_START := UINT#0;
		HEADER_STOP := UINT#0;
		BODY_START := UINT#0;
		BODY_STOP := UINT#0;
		HTTP_STATUS := '';
		ERROR := DWORD#0;
		ip_state := BYTE#1; (* Anmelden *)
		authentication := FALSE;
		delimiter2b := '$0D$0A';
		delimiter4b := '$0D$0A$0D$0A';

		(* LOGIN Parameter vorhanden *)
		(* LOGIN Parameter vorhanden *)
		IF URL_DATA.USER <> '' AND URL_DATA.PASSWORD <> '' THEN
			b64_str1 := CONCAT(URL_DATA.USER,':');
			b64_str1 := CONCAT(b64_str1,URL_DATA.PASSWORD); (* USER:PASSWORD *)
			b64_start := TRUE; (* BASE64 kodierung von Username *)
			authentication := TRUE;
			state := 5;
		ELSE
			state := 10;
		END_IF;
	        	(*####################  DEBUG-MESSAGE  ###################################*)
		(*IF _debug_enable THEN
	       		LOG_CL.NEW_MSG := 'HTTP: S00 START /IP_ID ~4';
	            	LOG_CL.PRINTF[4]  := BYTE_TO_STRING(IP_ID);
	            	LOG_MSG();
	        	END_IF;*)
	        	(*########################################################################*)
	END_IF;

5:	IF b64_start AND b64_done THEN (* warten auf base64 konvertierung *)
		b64_start := FALSE;
		state := 10;
	END_IF;

10:	IF ip_state = BYTE#3 THEN (* Bei IP_Control anmelden und auf freigabe warten *)
		idx := 0;
		text := CONCAT('GET ',URL_DATA.PATH);
		OSCAT_BASIC._STRING_TO_BUFFER(STR:=text,POS:=idx,PT:=ADR(S_BUF.BUFFER),SIZE:=SIZEOF(S_BUF.BUFFER)); (* GET path in buffer kopieren *)
		idx := idx + LEN(text);

		IF LEN(URL_DATA.QUERY) > 0 THEN
			S_BUF.BUFFER[idx] := 63; (* ASCII '?' *)
			idx := idx + 1;
			OSCAT_BASIC._STRING_TO_BUFFER(STR:=URL_DATA.QUERY,POS:=idx,PT:=ADR(S_BUF.BUFFER),SIZE:=SIZEOF(S_BUF.BUFFER)); (* QUERY in buffer kopieren *)
			idx := idx + LEN(URL_DATA.QUERY);
		END_IF;

		IF MODE >= BYTE#2 THEN (* gewünschte HTTP Version uebergeben *)
			text := ' HTTP/1.1';
		ELSE
			text := ' HTTP/1.0';
		END_IF;
		text := CONCAT(text,delimiter2b);
		OSCAT_BASIC._STRING_TO_BUFFER(STR:=text,POS:=idx,PT:=ADR(S_BUF.BUFFER),SIZE:=SIZEOF(S_BUF.BUFFER)); (* HTTP Version in buffer kopieren *)
		idx := idx + LEN(text);

		IF MODE = BYTE#1 THEN (* HTTP/1.0 mit persistenter Verbindung gewünscht *)
			text := CONCAT('Connection: Keep-Alive',delimiter2b); (* workaround für pcworx -> kein $0D$0A als Stringkonstante möglich *)
		ELSIF MODE = BYTE#3 THEN (* HTTP/1.1 ohne persistenter Verbindung gewünscht *)
			text := CONCAT('Connection: Close',delimiter2b); (* workaround für pcworx -> kein $0D$0A als Stringkonstante möglich *)
		ELSE
			text := '';
		END_IF;

		(* Zusatz Parameter übernehmen *)
		text := CONCAT(text,URL_DATA.HEADER);
		OSCAT_BASIC._STRING_TO_BUFFER(STR:=text,POS:=idx,PT:=ADR(S_BUF.BUFFER),SIZE:=SIZEOF(S_BUF.BUFFER)); (* HTTP Version in buffer kopieren *)
		idx := idx + LEN(text);

		IF authentication THEN
			text := CONCAT('Authorization: Basic ',b64_str2);
			text := CONCAT(text,delimiter2b); (* workaround für pcworx -> kein $0D$0A als Stringkonstante möglich *)
			OSCAT_BASIC._STRING_TO_BUFFER(STR:=text,POS:=idx,PT:=ADR(S_BUF.BUFFER),SIZE:=SIZEOF(S_BUF.BUFFER)); (* HTTP Host in buffer kopieren *)
			idx := idx + LEN(text);
		END_IF;

		text := CONCAT('Host: ',URL_DATA.DOMAIN);
		text := CONCAT(text,delimiter4b); (* workaround für pcworx -> kein $0D$0A als Stringkonstante möglich *)
		OSCAT_BASIC._STRING_TO_BUFFER(STR:=text,POS:=idx,PT:=ADR(S_BUF.BUFFER),SIZE:=SIZEOF(S_BUF.BUFFER)); (* HTTP Host in buffer kopieren *)
		idx := idx + LEN(text);

		(* IP Datenverkehr einrichten *)
		IF FIND(';HTTPS;https;Https;', CONCAT(URL_DATA.PROTOCOL,';')) > 1 THEN
			IP_C.C_PORT := SEL(URL_DATA.PORT = WORD#0,URL_DATA.PORT,WORD#443); (* Portnummer eintragen *)
			IP_C.MAILBOX[16] := BYTE#1; (* SSL Mode freigeben *)
		ELSE
			IP_C.C_PORT := SEL(URL_DATA.PORT = WORD#0,URL_DATA.PORT,WORD#80);  (* Portnummer eintragen *)
		END_IF;

		IP_C.C_IP := ip4_stored; (* IP eintragen *)
		IP_C.C_MODE := BYTE#0; (* Mode: TCP+AKTIV+PORT+IP *)
		IP_C.C_ENABLE := TRUE; (* Verbindungsaufbau freigeben *)
		IP_C.TIME_RESET := TRUE; (* Zeitueberwachung rücksetzen *)
		IP_C.R_OBSERVE := TRUE; (* Datenempfang ueberwachen *)
		S_BUF.SIZE := INT_TO_UINT(idx); (* Sendelänge eintragen *)
		R_BUF.SIZE := UINT#0; (* Empfangslänge rücksetzen *)

		state := 30;
	        	(*####################  DEBUG-MESSAGE  ###################################*)
	        	(*IF _debug_enable THEN
	        		LOG_CL.NEW_MSG := 'HTTP: S20 SEND /IP_ID ~4';
	            	LOG_CL.PRINTF[4]  := BYTE_TO_STRING(IP_ID);
	            	LOG_MSG();
	        	END_IF;*)
	        	(*########################################################################*)
	END_IF;

30:	rcv_timeout := (IP_C.ERROR AND DWORD#16#0000_FF00) = DWORD#16#0000_FF00;
	con_rdce :=     (IP_C.ERROR AND DWORD#16#FD00_0000) = DWORD#16#FD00_0000;

	IF S_BUF.SIZE = UINT#0 THEN
		IF total_size = 0 THEN
			IF R_BUF.SIZE > UINT#15 THEN; (* länge der empfangenen Daten prüfen *)

				(* HTTP HEADER Ende suchen -> durch $0D$A$0D$A erkennbar bei DEC RT-11,CP/M,MS-DOS,Windows *)
				del_end := '$0D$0A$0D$0A';
				del_pos := OSCAT_BASIC.BUFFER_SEARCH(PT:=ADR(R_BUF.BUFFER),SIZE:=R_BUF.SIZE,STR:=del_end,POS:=0,IGN:=FALSE);

				(* kein Ende gefunden ? -> andere Ende-Codierung suchen *)
				IF del_pos = 0 THEN
					del_end := '$0A$0A';
					(* HTTP HEADER Ende suchen -> durch $0A$0A erkennbar bei Multics, Unix-Derivate,Mac OS X *)
					del_pos := OSCAT_BASIC.BUFFER_SEARCH(PT:=ADR(R_BUF.BUFFER),SIZE:=R_BUF.SIZE,STR:=del_end,POS:=0,IGN:=FALSE);
				END_IF;

				IF del_pos > 0 THEN
					HEADER_START := UINT#0;
					HEADER_STOP := INT_TO_UINT(del_pos + LEN(del_end) - 1);
					TOTAL_SIZE := -1; (* HTTP Header empfangen aber noch keine gesamtlänge bekannt *)
				END_IF;
		                	(*####################  DEBUG-MESSAGE  ###################################*)
		                	(*IF _debug_enable THEN
		                   	LOG_CL.NEW_MSG := 'HTTP: S20 HEADER_START ~1 / HEADER_STOP ~2/IP_ID ~4';
		                   	LOG_CL.PRINTF[4]  := BYTE_TO_STRING(IP_ID);
		                   	LOG_CL.PRINTF[1]  := UINT_TO_STRING(HEADER_START);
		                   	LOG_CL.PRINTF[2]  := UINT_TO_STRING(HEADER_STOP);
		                   	LOG_MSG();
		                	END_IF;*)
		                	(*########################################################################*)

				(* HTTP Statuscode auswerten: (kann 1.0 oder 1.1 sein *)
				READ_HTTP(size:=HEADER_STOP,pos:=0,SRC:='',pt:=R_BUF.BUFFER);

				i := LEN(READ_HTTP.READ_HTTP);
				IF i > 7 THEN
					(* HTTP Version von HOST auswerten 1.0 oder 1.1 *)
					text:=MID(READ_HTTP.READ_HTTP,1,3);
					http_1_1_host := text = '1';

					(* Code und Meldung isolieren *)
					HTTP_STATUS := RIGHT(READ_HTTP.READ_HTTP,i-4);
				END_IF;

				(* positive HTTP Anfrage ? *)
				IF FIND(HTTP_STATUS,'200') > 0 THEN

					(* 'Content-Length: Wert einlesen auswerten *)
					READ_HTTP(size:=HEADER_STOP,pos:=0,SRC:='CONTENT-LENGTH',pt:=R_BUF.BUFFER);
					text:=READ_HTTP.READ_HTTP;

					IF LEN(text) >= 1 THEN
						IF OSCAT_BASIC.IS_NUM(str:=text) THEN
							(* erwartete gesamtmenge an Bytes berechnen *)
							total_size := STRING_TO_INT(text) + UINT_TO_INT(HEADER_STOP) + 1;
                           					(*####################  DEBUG-MESSAGE  ###################################*)
                           					(*IF _debug_enable THEN
                              					LOG_CL.NEW_MSG := 'HTTP: S20 HEADER ~1, BODY ~2 TOTAL ~3 /IP_ID ~4';
                             					LOG_CL.PRINTF[4]  := BYTE_TO_STRING(IP_ID);
                               					LOG_CL.PRINTF[1]  := UINT_TO_STRING(HEADER_STOP);
                               					LOG_CL.PRINTF[2]  := INT_TO_STRING(TOTAL_SIZE-UINT_TO_INT(HEADER_STOP));
                               					LOG_CL.PRINTF[3]  := INT_TO_STRING(TOTAL_SIZE);
                              					LOG_MSG();
                          					END_IF;*)
                          					(*########################################################################*)
						END_IF;
					END_IF;
				ELSE
					ERROR := DWORD#16#000000FC; (* Fehler durch HTTP-Statuscodes *)
				END_IF;
			END_IF;
		(* 1. bei bekannter Content-Length wird nach erhalt der erwartenen Daten die verbindung beendet *)
		(* 2. bei persistenter Verbindung muss bei unbekannter Datenmenge auf Receive-Timeout gewartet werden *)
		(* 3. wenn nach datenempfang die verbindung vom host unterbrochen wird *)
		ELSIF (R_BUF.SIZE >= INT_TO_UINT(total_size)) OR
			(R_BUF.SIZE > UINT#0 AND total_size < 0 AND ((rcv_timeout OR con_rdce) OR (IP_C.C_STATE = BYTE#1))) THEN

			IF R_BUF.SIZE - 1 > HEADER_STOP THEN (* BODY Daten vorhanden *)
				BODY_START := HEADER_STOP + UINT#1;
				BODY_STOP := R_BUF.SIZE - 1;
		                	(*####################  DEBUG-MESSAGE  ###################################*)
		                	(*IF _debug_enable THEN
		                   	LOG_CL.NEW_MSG := 'HTTP: S20 BODY ~1, START ~2 END ~3 /IP_ID ~4';
		                   	LOG_CL.PRINTF[4]  := BYTE_TO_STRING(IP_ID);
		                   	LOG_CL.PRINTF[1]  := UINT_TO_STRING(HEADER_STOP);
		                   	LOG_CL.PRINTF[2]  := UINT_TO_STRING(BODY_START);
		                   	LOG_CL.PRINTF[3]  := UINT_TO_STRING(BODY_STOP);
		                   	LOG_MSG();
		               	END_IF;*)
		               	(*########################################################################*)
			END_IF;

			DONE := TRUE;
			IP_C.C_ENABLE := FALSE; (* Verbindung abbauen *)
			state := 40;
            		(*####################  DEBUG-MESSAGE  ###################################*)
            		(*IF _debug_enable THEN
                			LOG_CL.NEW_MSG := 'HTTP: S30 OK /IP_ID ~4';
                			LOG_CL.PRINTF[4]  := BYTE_TO_STRING(IP_ID);
                			LOG_MSG();
            		END_IF;*)
            		(*########################################################################*)
		END_IF;
	END_IF;

	IF IP_C.ERROR <> DWORD#0 THEN
		(* bei unbekannter Content-size ist nicht bekannt ob bzw wieviele Telegramme noch folgen werden *)
		(* darum wird nach receive-timeout oder Remote disconnect error der fehler wieder ausgefiltert (logischer fehler) *)
		IF rcv_timeout AND DONE THEN
			IP_C.ERROR := IP_C.ERROR AND DWORD#16#FFFF_00FF; (* Fehler wieder rücksetzen *)
		ELSIF con_rdce AND DONE THEN
			IP_C.ERROR := IP_C.ERROR AND DWORD#16#00FF_FFFF; (* Fehler wieder rücksetzen *)
		ELSE
			ERROR := IP_C.ERROR;
		END_IF;
	END_IF;

	IF ERROR > DWORD#0 THEN
		IP_C.C_ENABLE := FALSE; (* Verbindungsaufbau sperren *)
		state := 40;
	        	(*####################  DEBUG-MESSAGE  ###################################*)
	        	(*IF _debug_enable THEN
	            	LOG_CL.NEW_MSG := 'HTTP: S30 ERROR ~1 /IP_ID ~4';
	            	LOG_CL.PRINTF[1]  := DWORD_TO_STRING(ERROR);
	            	LOG_CL.PRINTF[4]  := BYTE_TO_STRING(IP_ID);
	            	LOG_MSG();
	        	END_IF;*)
	        	(*########################################################################*)
	END_IF;

40:	IF (UNLOCK_BUF OR NOT DONE) THEN (* Warten auf Release und Verbindung beendet -> IP_ID vom Stack nehmen *)
		IP_STATE := BYTE#4; (* Abmelden *)
		DONE := FALSE;
		IP_C.MAILBOX[16] := BYTE#0; (* SSL Mode beenden *)
		state := 0;
	END_IF;
END_CASE;

get_last := GET; (* letzten Status sichern zur Flankenerkennung *)

IP_FIFO(FIFO:=IP_C.FIFO,STATE:=ip_state,ID:=ip_id); (* IP_FIFO *)

BASE64_ENCODE_STR(RUN:=b64_start,STR1:=b64_str1,STR2:=b64_str2); (* BASE64 kodierung *)
b64_done:=BASE64_ENCODE_STR.DONE;

(*####################  DEBUG-MESSAGE  ###################################*)
(*IF _debug_enable THEN
	IF state <> _debug_state_last THEN
		LOG_CL.NEW_MSG := 'http_get: /last ~1 /New ~2';
		LOG_CL.PRINTF[1] := INT_TO_STRING(_debug_state_last);
		LOG_CL.PRINTF[2] := INT_TO_STRING(state);
		LOG_MSG();
		_debug_state_last := state;
	END_IF;
END_IF;*)
(*########################################################################*)

(* revision history
ks	18. oct. 2008	rev 1.0
	original version

ks	20. oct. 2009	rev 1.1
	Fehler bei body-suche bei $0a$0a korrigiert,Codeoptimierung,
	new VAR del_pos , del_end (Networkbuffer und Buffer-funktionen auf Basis 0)

ks	28. oct. 2009	rev 1.2
	über url.header können zusätzliche header-infos übergeben werden

ks	12. apr. 2011	rev 1.3
	verbesserte fehlererkennung und fehlerkorrektur bei buffer_to_string

ks	31. mar. 2016	rev 1.4
	Authentication und SSL (HTTPS) hinzugefügt, DONE später zurücksetzen

*)

END_FUNCTION_BLOCK

// POUs/NETWORK/READ_HTTP
FUNCTION_BLOCK READ_HTTP
VAR_INPUT
	SIZE : UINT;
	POS : INT;
	SRC : STRING;
END_VAR
VAR_IN_OUT
	PT : NW_BUF_LONG;
END_VAR
VAR_OUTPUT
	READ_HTTP : STRING(OSCAT_BASIC.STRING_LENGTH);
END_VAR
VAR
	index : INT;
	s1 : INT;
	e1 : INT;
	stop : INT;
END_VAR

(*

version 1.1 20. oct. 2009
programmer 	ks
tested by	ks

READ_HTTP wertet die Informationen einer HTTP-Request aus, und stellt die Daten zu Verfügung.
*)

stop := UINT_TO_INT(SIZE) - 1;

IF LEN(SRC) = 0 THEN
	(* wenn kein Suchbegriff vorhanden ist, dann den HTTP-STATUS auswerten *)
	SRC := 'HTTP/'; (* neuer Suchbegriff *)
ELSE
	(* gesuchten Parametertext ergänzen *)
	SRC := CONCAT(SRC,': ');
END_IF;

s1 := OSCAT_BASIC.BUFFER_SEARCH(pt:=ADR(PT),SIZE:=SIZE,STR:=SRC,POS:=POS,IGN:=TRUE);

IF s1 >= 0 THEN (* Text found *)
	e1 := s1;

	(* search start of line *)
	index := s1 - 1;
	WHILE (index > 0) DO
		IF pt[index] < BYTE#32 THEN EXIT; END_IF;
		s1 := s1 - 1;
		index := index - 1;
	END_WHILE;

	(* search end of line *)
	index := e1 + 1;
	WHILE (index <= stop) DO
		IF pt[index] < BYTE#32 THEN EXIT; END_IF;
		e1 := e1 + 1;
		index := index + 1;
	END_WHILE;

	s1 := s1 + LEN(SRC); (* 'suchbegriff: ' nicht mitkopieren *)

	(* copy string *)
	READ_HTTP := OSCAT_BASIC.BUFFER_TO_STRING(PT:=ADR(PT),SIZE:=SIZE,START:=s1,STOP:=e1);
ELSE
	READ_HTTP := '';
END_IF;

(* revision history

ks	18. oct. 2008	rev 1.0
	original version

ks	20. oct. 2009	rev 1.1
	Networkbuffer und Buffer-funktionen auf Basis 0

*)

END_FUNCTION_BLOCK

// POUs/NETWORK/DNS_DYN
FUNCTION_BLOCK DNS_DYN
VAR_IN_OUT
	IP_C : IP_C; (* IP_Control Verwaltungsstruktur *)
	S_BUF : NETWORK_BUFFER;
	R_BUF : NETWORK_BUFFER;
END_VAR
VAR_INPUT
	ENABLE : BOOL;
	UPDATE : BOOL;
	T_UPDATE : TIME := T#1h;
	MODE : BYTE;
	HOSTNAME : STRING(30);
	USERNAME : STRING(20);
	PASSWORD : STRING(20);
	IP4 : DWORD;
END_VAR
VAR_OUTPUT
	BUSY : BOOL;
	DONE : BOOL;
	ERROR_C : DWORD;
	ERROR_T : BYTE;
END_VAR
VAR
	DNS_CLIENT : DNS_CLIENT;
	HTTP_GET : HTTP_GET;
	BASE64_ENCODE_STR : BASE64_ENCODE_STR;
	URL_DATA : url;
	update_last : BOOL;
	state : INT;
	base64_done : BOOL;
	s1 : STRING(144);
	s2 : STRING(192);
	w : TON;
END_VAR

(*

version 1.2		02. dec. 2009
programmer 		ks
tested by		ks

YAHOO_WEATHER lädt vom Yahoo-Webserver einen Wetter RSS-Feed und analysiert die Daten und legt diese in einem Array ab
*)

CASE state OF

00:	IF ENABLE AND ((UPDATE AND NOT update_last) OR w.Q) THEN
		state := 20;
		DONE := FALSE;
		BUSY := TRUE;
		ERROR_C := DWORD#0;
		ERROR_T := BYTE#0;

		IF MODE = 0 THEN (* dyndns.org *)
			s2 := CONCAT('http://members.dyndns.org/nic/update?hostname=',HOSTNAME);
		ELSE (* selfhost.de *)
			s2 := 'http://carol.selfhost.de/nic/update?hostname=1';
		END_IF;
		IF IP4 > 0 THEN (* parametrierte IP verwenden *)
			s1 := CONCAT('&myip=',IP4_TO_STRING(IP4));
			s2 := CONCAT(s2,s1);
		END_IF;
		URL_DATA:=STRING_TO_URL(STR:=s2, DEFAULT_PROTOCOL:='', DEFAULT_PATH:=''); (* URL for DNS UND HTTP-GET *)
		s1 := CONCAT(USERNAME,':');
		s1 := CONCAT(s1,PASSWORD); (* BASE64 Encode Text *)
	END_IF;

20:	IF DNS_CLIENT.DONE THEN (* DNS_CLIENT *)
			state := 40;
	ELSIF (DNS_CLIENT.ERROR > DWORD#00) THEN (* Fehlerbehandlung *)
		ERROR_C := DNS_CLIENT.ERROR;
		ERROR_T := BYTE#01;
		BUSY := FALSE;
		state := 0;
	END_IF;

40: IF base64_done THEN (* BASE64 Encode beendet ? *)
		s1 := CONCAT('Authorization: Basic ',s2);
		s1 := CONCAT(s1,'$0D$0AUser-Agent: x$0D$0A');
		URL_DATA.HEADER := s1;
		state := 60;
	END_IF;

60:	IF HTTP_GET.DONE THEN
		state := 0;
		BUSY := FALSE;
		DONE := TRUE;

		(* !! Codes !!
		Successful Updates: 		good , nchg
		Update Syntax Errors:		badsys , badagent
		Account-Related Errors:		badauth , !donator
		Hostname-Related Errors:	notfqdn , nohost , !yours , numhost , abuse
		Server Error Conditions:	dnserr , 911
		*)
		s2 := OSCAT_BASIC.BUFFER_TO_STRING(PT:=ADR(R_BUF.BUFFER),SIZE:=SIZEOF(R_BUF.BUFFER),START:=HTTP_GET.BODY_START + 3,STOP:=HTTP_GET.BODY_STOP - 7);
		IF FIND(s2,'good') = 0 THEN
			IF FIND(s2,'nochg') = 0 THEN
				ERROR_C := DWORD#1;
				ERROR_T := BYTE#03;
				DONE := FALSE;
			END_IF;
		END_IF;
	ELSIF (HTTP_GET.ERROR > DWORD#00) THEN (* Fehlerbehandlung *)
		ERROR_C := HTTP_GET.ERROR;
		ERROR_T := BYTE#02;
		BUSY := FALSE;
		state := 0;
	END_IF;

END_CASE;

DNS_CLIENT(IP_C:=IP_C,	S_BUF:=S_BUF, R_BUF:=R_BUF,DOMAIN:=URL_DATA.DOMAIN, IP4_DNS:=0, ACTIVATE:=state=20); (* DNS_CLIENT *)
HTTP_GET( IP_C:=IP_C, S_BUF:=S_BUF, R_BUF:=R_BUF, IP4:=DNS_CLIENT.IP4, GET:=state=60, MODE:=2, UNLOCK_BUF:=state<>60,URL_DATA:=URL_DATA); (* HTTP_GET *)
BASE64_ENCODE_STR( RUN:=state=40, STR1:=s1, STR2:=s2, DONE=>base64_done); (* BASE64 Encode *)

IF T_UPDATE > T#0ms THEN w(IN:=state=0, PT:=T_UPDATE); END_IF;
update_last := UPDATE;

(* revision history
ks	01. jan. 2010	rev 1.0
	original version

*)

END_FUNCTION_BLOCK

// POUs/WEATHER/YAHOO_WEATHER
FUNCTION_BLOCK YAHOO_WEATHER
VAR_IN_OUT
	IP_C : IP_C; (* IP_Control Verwaltungsstruktur *)
	S_BUF : NETWORK_BUFFER;
	R_BUF : NETWORK_BUFFER;
	YW : YAHOO_WEATHER_DATA;
END_VAR
VAR_INPUT
	ACTIVATE : BOOL;
	UNITS : BOOL;
	LOCATION : STRING(20);
END_VAR
VAR_OUTPUT
	BUSY : BOOL;
	DONE : BOOL;
	ERROR_C : DWORD;
	ERROR_T : BYTE;
END_VAR
VAR
	CTRL : XML_CONTROL;
	XML_READER : XML_READER;
	URL_DATA : url;
	DNS_CLIENT : DNS_CLIENT;
	HTTP_GET : HTTP_GET;
	activate_last : BOOL;
	value_int : INT;
	value_real : REAL;
	v_real : REAL;
	state : INT;
	cycle : INT;
	day_idx :	INT;
	idx : INT;
	cnt :	INT;
	repeat_request : BOOL;
	repeat_wait_time : UDINT := 5000; (* Repeat-Waittime *)
	repeat_count : USINT;
	repeat_max_count : USINT := 3;	(* maximal repeat *)
	repeat_tx : UDINT;
	tx : UDINT;

	(*
	_debug_state_last : INT := -1;
	_debug_enable : BOOL := TRUE;
	LOG_MSG : LOG_MSG;
	*)

END_VAR

(*

version 1.6		22. may. 2017
programmer 		ks
tested by			ks

YAHOO_WEATHER lädt vom Yahoo-Webserver einen Wetter RSS-Feed und analysiert die Daten und legt diese in einem Array ab
*)

(* read system time *)
tx := OSCAT_BASIC.T_PLC_MS();

CASE state OF

00:	IF ACTIVATE AND NOT activate_last THEN
		state := 40;
		DONE := FALSE;
		BUSY := TRUE;
		ERROR_C := DWORD#0;
		ERROR_T := BYTE#0;
		cycle := 0;
		repeat_count := USINT#0;
		repeat_request := FALSE;
  		URL_DATA.DOMAIN := 'query.yahooapis.com'; (* Domainname für DNS_CLIENT *)
	END_IF;

40:	IF DNS_CLIENT.DONE THEN
		state := 50;
	ELSIF (DNS_CLIENT.ERROR > DWORD#00) THEN
		(* Fehlerbehandlung *)
		ERROR_C := DNS_CLIENT.ERROR;
		ERROR_T := BYTE#01;
		state   := 100;
	END_IF;

50:   	(* Teil 1: http://query.yahooapis.com/v1/public/yql?q=select%20units,wind,atmosphere,astronomy,location%20from%20weather.forecast%20where%20woeid=551801%20AND%20u=%27c%27
             Teil 2: http://query.yahooapis.com/v1/public/yql?q=select%20item%20from%20weather.forecast%20where%20woeid=551801%20AND%20u=%27c%27 *)

	IF cycle = 0 THEN
  		URL_DATA.QUERY := 'q=select%20units,wind,atmosphere,astronomy,location%20from%20weather.forecast%20where%20woeid='; (* Teil 1 - infos *)
  	ELSE
  		URL_DATA.QUERY := 'q=select%20item%20from%20weather.forecast%20where%20woeid='; (* Teil 2 - Tagesdaten *)
  	END_IF;

  	URL_DATA.QUERY := CONCAT(URL_DATA.QUERY,LOCATION); (* location *)

  	IF UNITS THEN
    		URL_DATA.QUERY := CONCAT(URL_DATA.QUERY,'%20and%20u=%27f%27'); (* fahrenheit *)
  	ELSE
    		URL_DATA.QUERY := CONCAT(URL_DATA.QUERY,'%20and%20u=%27c%27'); (* celsius *)
  	END_IF;

  	URL_DATA.PATH := '/v1/public/yql';

  	state := 60;

60:	IF HTTP_GET.DONE THEN
		state := 80;
		CTRL.START_POS := HTTP_GET.BODY_START;
		CTRL.STOP_POS := HTTP_GET.BODY_STOP;
		CTRL.COMMAND := WORD#2#10000000_00011000; (* ONLY TEXT AND ATTRIBUTE *)
		CTRL.WATCHDOG  := T#1ms;

	ELSIF (HTTP_GET.ERROR > DWORD#00) THEN
		(* Fehlerbehandlung *)
		ERROR_C := HTTP_GET.ERROR;
		ERROR_T := BYTE#02;
		state := 100;
	END_IF;

80: XML_READER(CTRL:=CTRL,BUF:=R_BUF.BUFFER); (* XML Daten seriell lesen *)
	IF CTRL.TYP < 98 THEN (* nur auswerten wenn kein Watchdog durchlauf *)
		value_int := 0;
		value_real := 0.0;
		(* automatische konvertierung in real und int ausführen *)
		IF LEN(CTRL.VALUE) <= 20 THEN
			v_real:=OSCAT_BASIC.FLOAT_TO_REAL(FLT:=CTRL.VALUE);
			IF OSCAT_BASIC.CHK_REAL(v_real) = 0 THEN (* !!! prüft auf gültigen REAL Wert, ansonsten kann Twincat 2.x abstürzen !!!!  *)
				value_real := v_real;
				value_int := REAL_TO_INT(value_real);
			END_IF;
		END_IF;

		(*####################  DEBUG-MESSAGE  ###################################*)
		(*IF _debug_enable THEN
			LOG_CL.NEW_MSG := 'XML: ~2 # ~3 # ~4 # ~5';
			LOG_CL.PRINTF[2] := UINT_TO_STRING(CTRL.LEVEL);
			LOG_CL.PRINTF[3] := UINT_TO_STRING(CTRL.COUNT);
			LOG_CL.PRINTF[4] := CTRL.ELEMENT;
			LOG_CL.PRINTF[5] := CTRL.VALUE;
			LOG_MSG();
		END_IF;*)
		(*########################################################################*)

		(* Antwortdaten stehen noch nicht bereit -> Warten und Abfrage wiederholen *)
		IF ctrl.COUNT = 7 AND (ctrl.VALUE = '0')  THEN

			repeat_count := repeat_count + USINT#1;

			(* maximale Anzahl an Wiederholungen erreicht -> Mit Fehler abbrechen *)
			IF repeat_count > repeat_max_count THEN

				(* Fehlerbehandlung *)
				ERROR_C := USINT_TO_DWORD(repeat_max_count);
				ERROR_T := BYTE#03;
				state   := 100;

			ELSE
				repeat_request := TRUE;
				state := 100;

				(*####################  DEBUG-MESSAGE  ###################################*)
				(*IF _debug_enable THEN
					LOG_CL.NEW_MSG := 'Request Error  / Part ~2 / Count ~3';
					LOG_CL.PRINTF[2] := INT_TO_STRING(cycle);
					LOG_CL.PRINTF[3] := USINT_TO_STRING(repeat_count);
					LOG_MSG();
				END_IF;*)
				(*########################################################################*)

			END_IF;

		END_IF;

		IF cycle = 0 THEN
	      		(* ------------ Teil 1 --------------*)
	      		CASE UINT_TO_INT(CTRL.COUNT) OF
	        		014: YW.location_city := CTRL.VALUE;
	        		015: YW.location_country := CTRL.VALUE;
	        		016: YW.location_region := CTRL.VALUE;
	        		020: YW.wind_chill := value_int;
	        		021: YW.wind_direction := value_int;
	        		022: YW.wind_speed := value_real;
	        		026: YW.atmosphere_humidity := value_int;
	        		027: YW.atmosphere_pressure := value_real;
	        		028: YW.atmosphere_rising := value_int;
	        		029: YW.atmosphere_visibility := value_real;
	        		033: YW.astronomy_sunrise := CTRL.VALUE;
	        		034: YW.astronomy_sunset := CTRL.VALUE;
	        		038: YW.unit_distance := CTRL.VALUE;
	        		039: YW.unit_pressure := CTRL.VALUE;
	        		040: YW.unit_speed := CTRL.VALUE;
	        		041: YW.unit_temperature := CTRL.VALUE;
	      		END_CASE;
	    	ELSE
	      		(* ------------ Teil 2 --------------*)
	      		CASE UINT_TO_INT(CTRL.COUNT) OF
	        		018: YW.GEO_LATITUDE := value_real;
	        		022: YW.GEO_LONGITUDE := value_real;
	
			032: YW.CUR_CONDITIONS_CODE := value_int;
			         YW.CUR_CONDITIONS_ICON := value_int;
	        		034: YW.CUR_CONDITIONS_TEMP := value_int;
	        		035: YW.CUR_CONDITIONS_TEXT := CTRL.VALUE;
	
			039: YW.FORECAST_TODAY_CODE := value_int;
			         YW.FORECAST_TODAY_ICON := value_int;
			040: YW.FORECAST_TODAY_DATE_LONG := CTRL.VALUE;
	        		042: YW.FORECAST_TODAY_HIGH_TEMP := value_int;
	        		043: YW.FORECAST_TODAY_LOW_TEMP := value_int;
	        		044: YW.FORECAST_TODAY_TEXT := CTRL.VALUE;

			048..125: (* forcast day 1-10 *)
				cnt := UINT_TO_INT(CTRL.COUNT) - 48;
				day_idx := cnt / 9 + 1;
				idx := cnt MOD 9;
	      	  		CASE idx OF
					0:	YW.FORECAST_DAY[day_idx].CODE := value_int;
						YW.FORECAST_DAY[day_idx].ICON := value_int;
					1:	YW.FORECAST_DAY[day_idx].DATE_LONG := CTRL.VALUE;
					3:	YW.FORECAST_DAY[day_idx].HIGH_TEMP := value_int;
					4:	YW.FORECAST_DAY[day_idx].LOW_TEMP := value_int;
					5:	YW.FORECAST_DAY[day_idx].TEXT := CTRL.VALUE;
	      	  		END_CASE;
	      		END_CASE;
	    	END_IF;
	ELSIF CTRL.TYP = 99 THEN (* EXIT - letztes Element gelesen *)
		state := 100;
	END_IF;

100:	(* UNLOCK HTTP DATA *)
	IF (NOT HTTP_GET.DONE) THEN

		IF repeat_request THEN
			repeat_tx := tx;
    			state := 110;

		ELSIF cycle = 0 AND ERROR_T = BYTE#0 THEN
			(* Teil 2 ausführen *)
    			state := 50;
			cycle := cycle + 1;
			repeat_count := USINT#0;
		ELSE
	    		state := 0;
	    		BUSY  := FALSE;
	    		DONE := ERROR_T = BYTE#0;
		END_IF;
	END_IF;

110: (* REPEAT REQUEST - WAIT TIME *)
	IF tx > repeat_tx + repeat_wait_time THEN

